	{attribute 'TcIecLibraryType'}
	{attribute 'external_name' := 'F_VN_KeyPointsGFTTExp_GUID_AB658F05_AE08_576E_4247_1E7B0BCA6233'}
	(* Detects keypoints using the GFTT method, which detects strong corners. (expert function) *)
	FUNCTION F_VN_KeyPointsGFTTExp : HRESULT
	VAR_INPUT
		ipSrcImage	:	ITcVnImage;	(* Source image *)
		ipKeyPoints	:	REFERENCE TO ITcVnContainer;	(* Returns a container which is filled with the keypoints (ContainerType_Vector_TcVnKeyPoint; Non-zero interface pointers are reused.) *)
		ipMask	:	ITcVnImage;	(* Mask to specify, where to look for keypoints (set to 0 if no mask required) *)
		stParams	:	REFERENCE TO TcVnParamsGFTT;	(* Additional expert parameters *)
		hrPrev	:	HRESULT;	(* HRESULT indicating the result of previous operations (If SUCCEEDED(hrPrev) equals false, no operation is executed.) *)
	END_VAR

END_FUNCTION

// Functions/Keypoint Features/F_VN_KeyPointsMSER

	{attribute 'TcIecLibraryType'}
	{attribute 'external_name' := 'F_VN_KeyPointsMSER_GUID_593D7D5C_CD62_5D15_521E_85C3A9A2E7E5'}
	(* Detects keypoints using the MSER method. *)
	FUNCTION F_VN_KeyPointsMSER : HRESULT
	VAR_INPUT
		ipSrcImage	:	ITcVnImage;	(* Source image *)
		ipKeyPoints	:	REFERENCE TO ITcVnContainer;	(* Returns a container which is filled with the keypoints (ContainerType_Vector_TcVnKeyPoint; Non-zero interface pointers are reused.) *)
		hrPrev	:	HRESULT;	(* HRESULT indicating the result of previous operations (If SUCCEEDED(hrPrev) equals false, no operation is executed.) *)
	END_VAR

END_FUNCTION

// Functions/Keypoint Features/F_VN_KeyPointsMSERExp

	{attribute 'TcIecLibraryType'}
	{attribute 'external_name' := 'F_VN_KeyPointsMSERExp_GUID_ABE22F08_7F3B_521F_6B7B_35024442B7CC'}
	(* Detects keypoints using the MSER method. (expert function) *)
	FUNCTION F_VN_KeyPointsMSERExp : HRESULT
	VAR_INPUT
		ipSrcImage	:	ITcVnImage;	(* Source image *)
		ipKeyPoints	:	REFERENCE TO ITcVnContainer;	(* Returns a container which is filled with the keypoints (ContainerType_Vector_TcVnKeyPoint; Non-zero interface pointers are reused.) *)
		ipMask	:	ITcVnImage;	(* Mask to specify, where to look for keypoints (set to 0 if no mask required) *)
		stParams	:	REFERENCE TO TcVnParamsMSER;	(* Additional expert parameters *)
		hrPrev	:	HRESULT;	(* HRESULT indicating the result of previous operations (If SUCCEEDED(hrPrev) equals false, no operation is executed.) *)
	END_VAR

END_FUNCTION

// Functions/Keypoint Features/F_VN_KeyPointsSB

	{attribute 'TcIecLibraryType'}
	{attribute 'external_name' := 'F_VN_KeyPointsSB_GUID_2AF0CAD1_6515_5A1D_720D_33AA4C99BB05'}
	(* Detects keypoints using a Simple Blob method:
          - several iterations apply different thresholds to source image
          - connected components (blobs) are detected
          - the center and radius of the blobs are returned as keypoints *)
	FUNCTION F_VN_KeyPointsSB : HRESULT
	VAR_INPUT
		ipSrcImage	:	ITcVnImage;	(* Source image *)
		ipKeyPoints	:	REFERENCE TO ITcVnContainer;	(* Returns a container which is filled with the keypoints (ContainerType_Vector_TcVnKeyPoint; Non-zero interface pointers are reused.) *)
		hrPrev	:	HRESULT;	(* HRESULT indicating the result of previous operations (If SUCCEEDED(hrPrev) equals false, no operation is executed.) *)
	END_VAR

END_FUNCTION

// Functions/Keypoint Features/F_VN_KeyPointsSBExp

	{attribute 'TcIecLibraryType'}
	{attribute 'external_name' := 'F_VN_KeyPointsSBExp_GUID_81F47CE7_8C3F_532C_650C_F93B4893D1D6'}
	(* 
          Detects keypoints using a Simple Blob method (expert function)
          - several iterations apply different thresholds to source image
          - connected components (blobs) are detected
          - the center and radius of the blobs are returned as keypoints
         *)
	FUNCTION F_VN_KeyPointsSBExp : HRESULT
	VAR_INPUT
		ipSrcImage	:	ITcVnImage;	(* Source image *)
		ipKeyPoints	:	REFERENCE TO ITcVnContainer;	(* Returns a container which is filled with the keypoints (ContainerType_Vector_TcVnKeyPoint; Non-zero interface pointers are reused.) *)
		ipMask	:	ITcVnImage;	(* Mask to specify, where to look for keypoints (currently not supported, set to 0) *)
		stParams	:	REFERENCE TO TcVnParamsSB;	(* Several parameters to filter the detected blobs *)
		hrPrev	:	HRESULT;	(* HRESULT indicating the result of previous operations (If SUCCEEDED(hrPrev) equals false, no operation is executed.) *)
	END_VAR

END_FUNCTION

// Functions/Keypoint Features/F_VN_MatchDescriptorsBF

	{attribute 'TcIecLibraryType'}
	{attribute 'external_name' := 'F_VN_MatchDescriptorsBF_GUID_B3966293_F5E5_53ED_7EA9_8C1C568150F9'}
	(* Match descriptors using a brute force approach. *)
	FUNCTION F_VN_MatchDescriptorsBF : HRESULT
	VAR_INPUT
		ipQueryDescriptors	:	ITcVnImage;	(* Query descriptors *)
		ipTrainDescriptors	:	ITcVnImage;	(* Training descriptors *)
		ipMatches	:	REFERENCE TO ITcVnContainer;	(* Returns a container which is filled with the descriptor matches (ContainerType_Vector_TcVnDMatch; Non-zero interface pointers are reused.) *)
		hrPrev	:	HRESULT;	(* HRESULT indicating the result of previous operations (If SUCCEEDED(hrPrev) equals false, no operation is executed.) *)
	END_VAR

END_FUNCTION

// Functions/Keypoint Features/F_VN_MatchDescriptorsBFExp

	{attribute 'TcIecLibraryType'}
	{attribute 'external_name' := 'F_VN_MatchDescriptorsBFExp_GUID_428339F2_71AA_5944_450A_B44763AAACE5'}
	(* Match descriptors using a brute force approach. (expert function) *)
	FUNCTION F_VN_MatchDescriptorsBFExp : HRESULT
	VAR_INPUT
		ipQueryDescriptors	:	ITcVnImage;	(* Query descriptors *)
		ipTrainDescriptors	:	ITcVnImage;	(* Training descriptors *)
		ipMatches	:	REFERENCE TO ITcVnContainer;	(* Returns a container which is filled with the descriptor matches (ContainerType_Vector_TcVnDMatch; Non-zero interface pointers are reused.) *)
		ipMask	:	ITcVnImage;	(* Mask to specify permissable matches, i.e. query[i] can be matched with train[j] only if mask[i][j] != 0 (set to 0 if no mask required) *)
		eNormType	:	ETcVnNormalizationType;	(* Normalization type (only L1, L2, L2SQR, HAMMING, HAMMING2 supported). HAMMING2 should be used for ORB descriptors if the ORB nBriefPoints parameter is 3 or 4) *)
		bCrossCheck	:	BOOL;	(* If true, only consistent matches are returned, i.e. query->train and train->query detect the same match *)
		hrPrev	:	HRESULT;	(* HRESULT indicating the result of previous operations (If SUCCEEDED(hrPrev) equals false, no operation is executed.) *)
	END_VAR

END_FUNCTION

// Functions/Keypoint Features/F_VN_MatchDescriptorsFlannLsh

	{attribute 'TcIecLibraryType'}
	{attribute 'external_name' := 'F_VN_MatchDescriptorsFlannLsh_GUID_6A0861D1_F3ED_5BC5_5E07_F85811927297'}
	(* Match descriptors using a FLANN based approach with LSH index. *)
	FUNCTION F_VN_MatchDescriptorsFlannLsh : HRESULT
	VAR_INPUT
		ipQueryDescriptors	:	ITcVnImage;	(* Query descriptors *)
		ipTrainDescriptors	:	ITcVnImage;	(* Training descriptors *)
		ipMatches	:	REFERENCE TO ITcVnContainer;	(* Returns a container which is filled with the descriptor matches (ContainerType_Vector_TcVnDMatch; Non-zero interface pointers are reused.) *)
		hrPrev	:	HRESULT;	(* HRESULT indicating the result of previous operations (If SUCCEEDED(hrPrev) equals false, no operation is executed.) *)
	END_VAR

END_FUNCTION

// Functions/Keypoint Features/F_VN_MatchDescriptorsFlannLshExp

	{attribute 'TcIecLibraryType'}
	{attribute 'external_name' := 'F_VN_MatchDescriptorsFlannLshExp_GUID_A6B46D94_1077_5A28_49E0_938BA5777C1C'}
	(* Match descriptors using a FLANN based approach with LSH index. (expert function) *)
	FUNCTION F_VN_MatchDescriptorsFlannLshExp : HRESULT
	VAR_INPUT
		ipQueryDescriptors	:	ITcVnImage;	(* Query descriptors *)
		ipTrainDescriptors	:	ITcVnImage;	(* Training descriptors *)
		ipMatches	:	REFERENCE TO ITcVnContainer;	(* Returns a container which is filled with the descriptor matches (ContainerType_Vector_TcVnDMatch; Non-zero interface pointers are reused.) *)
		nTableNumber	:	UDINT;	(* Number of tables *)
		nKeySize	:	UDINT;	(* Key size *)
		nMultiProbeLevel	:	UDINT;	(* Multi-probe level *)
		nChecks	:	UDINT;	(* Maximum number of visited leafs when searching for neighbors *)
		hrPrev	:	HRESULT;	(* HRESULT indicating the result of previous operations (If SUCCEEDED(hrPrev) equals false, no operation is executed.) *)
	END_VAR

END_FUNCTION

// Functions/Keypoint Features/F_VN_MatchDescriptorsKnnBF

	{attribute 'TcIecLibraryType'}
	{attribute 'external_name' := 'F_VN_MatchDescriptorsKnnBF_GUID_032847F3_E5D2_5453_7642_ACD471D5C57D'}
	(* Match descriptors (k nearest neighbors) using a brute force approach. *)
	FUNCTION F_VN_MatchDescriptorsKnnBF : HRESULT
	VAR_INPUT
		ipQueryDescriptors	:	ITcVnImage;	(* Query descriptors *)
		ipTrainDescriptors	:	ITcVnImage;	(* Training descriptors *)
		ipMatches	:	REFERENCE TO ITcVnContainer;	(* Returns a container which is filled with the descriptor matches (ContainerType_Vector_Vector_TcVnDMatch; Non-zero interface pointers are reused.) *)
		nK	:	UDINT;	(* Amount of best matches to search for *)
		hrPrev	:	HRESULT;	(* HRESULT indicating the result of previous operations (If SUCCEEDED(hrPrev) equals false, no operation is executed.) *)
	END_VAR

END_FUNCTION

// Functions/Keypoint Features/F_VN_MatchDescriptorsKnnBFExp

	{attribute 'TcIecLibraryType'}
	{attribute 'external_name' := 'F_VN_MatchDescriptorsKnnBFExp_GUID_4F5F4687_0324_5F53_4ED1_15CF466AF469'}
	(* Match descriptors (k nearest neighbors) using a brute force approach. (expert function) *)
	FUNCTION F_VN_MatchDescriptorsKnnBFExp : HRESULT
	VAR_INPUT
		ipQueryDescriptors	:	ITcVnImage;	(* Query descriptors *)
		ipTrainDescriptors	:	ITcVnImage;	(* Training descriptors *)
		ipMatches	:	REFERENCE TO ITcVnContainer;	(* Returns a container which is filled with the descriptor matches (ContainerType_Vector_Vector_TcVnDMatch; Non-zero interface pointers are reused.) *)
		nK	:	UDINT;	(* Amount of best matches to search for *)
		ipMask	:	ITcVnImage;	(* Mask to specify permissable matches, i.e. query[i] can be matched with train[j] only if mask[i][j] != 0 (set to 0 if no mask required) *)
		bCompactResult	:	BOOL;	(* If true, matches vector does not contain entries for fully masked-out query descriptors *)
		eNormType	:	ETcVnNormalizationType;	(* Normalization type (only L1, L2, L2SQR, HAMMING, HAMMING2 supported). HAMMING2 should be used for ORB descriptors if the ORB nBriefPoints parameter is 3 or 4) *)
		bCrossCheck	:	BOOL;	(* If true, only consistent matches are returned, i.e. query->train and train->query detect the same match (only used if nK = 1) *)
		hrPrev	:	HRESULT;	(* HRESULT indicating the result of previous operations (If SUCCEEDED(hrPrev) equals false, no operation is executed.) *)
	END_VAR

END_FUNCTION

// Functions/Keypoint Features/F_VN_MatchDescriptorsKnnFlannLsh

	{attribute 'TcIecLibraryType'}
	{attribute 'external_name' := 'F_VN_MatchDescriptorsKnnFlannLsh_GUID_C8244361_8A2E_5422_786B_9C4704343BF2'}
	(* Match descriptors (k nearest neighbors) using a FLANN based approach with LSH index. *)
	FUNCTION F_VN_MatchDescriptorsKnnFlannLsh : HRESULT
	VAR_INPUT
		ipQueryDescriptors	:	ITcVnImage;	(* Query descriptors *)
		ipTrainDescriptors	:	ITcVnImage;	(* Training descriptors *)
		ipMatches	:	REFERENCE TO ITcVnContainer;	(* Returns a container which is filled with the descriptor matches (ContainerType_Vector_Vector_TcVnDMatch; Non-zero interface pointers are reused.) *)
		nK	:	UDINT;	(* Amount of best matches to search for *)
		hrPrev	:	HRESULT;	(* HRESULT indicating the result of previous operations (If SUCCEEDED(hrPrev) equals false, no operation is executed.) *)
	END_VAR

END_FUNCTION

// Functions/Keypoint Features/F_VN_MatchDescriptorsKnnFlannLshExp

	{attribute 'TcIecLibraryType'}
	{attribute 'external_name' := 'F_VN_MatchDescriptorsKnnFlannLshExp_GUID_C49C1B5A_C1AC_5443_653F_891B8408EDAA'}
	(* Match descriptors (k nearest neighbors) using a FLANN based approach with LSH index. (expert function) *)
	FUNCTION F_VN_MatchDescriptorsKnnFlannLshExp : HRESULT
	VAR_INPUT
		ipQueryDescriptors	:	ITcVnImage;	(* Query descriptors *)
		ipTrainDescriptors	:	ITcVnImage;	(* Training descriptors *)
		ipMatches	:	REFERENCE TO ITcVnContainer;	(* Returns a container which is filled with the descriptor matches (ContainerType_Vector_Vector_TcVnDMatch; Non-zero interface pointers are reused.) *)
		nK	:	UDINT;	(* Amount of best matches to search for *)
		nTableNumber	:	UDINT;	(* Number of tables *)
		nKeySize	:	UDINT;	(* Key size *)
		nMultiProbeLevel	:	UDINT;	(* Multi-probe level *)
		nChecks	:	UDINT;	(* Maximum number of visited leafs when searching for neighbors *)
		hrPrev	:	HRESULT;	(* HRESULT indicating the result of previous operations (If SUCCEEDED(hrPrev) equals false, no operation is executed.) *)
	END_VAR

END_FUNCTION

// Functions/Keypoint Features/F_VN_RegionsMSER

	{attribute 'TcIecLibraryType'}
	{attribute 'external_name' := 'F_VN_RegionsMSER_GUID_55741E50_BE33_5462_61F4_4C1E00297C7D'}
	(* Detects regions using the MSER method. *)
	FUNCTION F_VN_RegionsMSER : HRESULT
	VAR_INPUT
		ipSrcImage	:	ITcVnImage;	(* Source image *)
		ipRegions	:	REFERENCE TO ITcVnContainer;	(* Returns a container which is filled with the region points (ContainerType_Vector_Vector_TcVnPoint2_DINT; Non-zero interface pointers are reused.) *)
		ipBoundingBoxes	:	REFERENCE TO ITcVnContainer;	(* Returns a container which is filled with the region bounding boxes (ContainerType_Vector_TcVnRectangle_DINT; Non-zero interface pointers are reused.) *)
		hrPrev	:	HRESULT;	(* HRESULT indicating the result of previous operations (If SUCCEEDED(hrPrev) equals false, no operation is executed.) *)
	END_VAR

END_FUNCTION

// Functions/Keypoint Features/F_VN_RegionsMSERExp

	{attribute 'TcIecLibraryType'}
	{attribute 'external_name' := 'F_VN_RegionsMSERExp_GUID_E4887BE5_69AC_5ABE_40D6_3515223EBD0A'}
	(* Detects regions using the MSER method. (expert function) *)
	FUNCTION F_VN_RegionsMSERExp : HRESULT
	VAR_INPUT
		ipSrcImage	:	ITcVnImage;	(* Source image *)
		ipRegions	:	REFERENCE TO ITcVnContainer;	(* Returns a container which is filled with the region points (ContainerType_Vector_Vector_TcVnPoint2_DINT; Non-zero interface pointers are reused.) *)
		ipBoundingBoxes	:	REFERENCE TO ITcVnContainer;	(* Returns a container which is filled with the region bounding boxes (ContainerType_Vector_TcVnRectangle_DINT; Non-zero interface pointers are reused.) *)
		stParams	:	REFERENCE TO TcVnParamsMSER;	(* Additional expert parameters *)
		hrPrev	:	HRESULT;	(* HRESULT indicating the result of previous operations (If SUCCEEDED(hrPrev) equals false, no operation is executed.) *)
	END_VAR

END_FUNCTION

// Functions/Code Reading/F_VN_ReadBarcode

	{attribute 'TcIecLibraryType'}
	{attribute 'external_name' := 'F_VN_ReadBarcode_GUID_7EE00F83_82CC_5410_5E28_06AA8744DAB0'}
	(* Detect and interpret a 1d barcode within the provided image.
          Can be canceled by Watchdog. *)
	FUNCTION F_VN_ReadBarcode : HRESULT
	VAR_INPUT
		ipSrcImage	:	ITcVnImage;	(* Source image (USINT elements, 1 channel or 3 channel (3 channel input is expected to be RGB and internally converted to Gray)) *)
		ipDecodedData	:	REFERENCE TO ITcVnContainer;	(* Returns the decoded code (ContainerType_Vector_String_SINT) *)
		eBarcodeType	:	UDINT;	(* Types of barcode to search for (ETcVnBarcodeType) *)
		hrPrev	:	HRESULT;	(* HRESULT indicating the result of previous operations (If SUCCEEDED(hrPrev) equals false, no operation is executed.) *)
	END_VAR

END_FUNCTION

// Functions/Code Reading/F_VN_ReadBarcodeExp

	{attribute 'TcIecLibraryType'}
	{attribute 'external_name' := 'F_VN_ReadBarcodeExp_GUID_746E9938_9353_5E2C_6CDD_CD6CAD35E403'}
	(* Detect and interpret a 1d barcode within the provided image.
          Can be canceled by Watchdog. *)
	FUNCTION F_VN_ReadBarcodeExp : HRESULT
	VAR_INPUT
		ipSrcImage	:	ITcVnImage;	(* Source image (USINT elements, 1 channel or 3 channel (3 channel input is expected to be RGB and internally converted to Gray)) *)
		ipDecodedData	:	REFERENCE TO ITcVnContainer;	(* Returns the decoded code (ContainerType_Vector_String_SINT) *)
		ipContours	:	REFERENCE TO ITcVnContainer;	(* Returns the code positions as contours (ContainerType_Vector_Vector_TcVnPoint2_DINT) *)
		eBarcodeType	:	UDINT;	(* Types of barcode to search for (ETcVnBarcodeType) *)
		nCodeNumber	:	DINT;	(* Number of 1d barcode that should be detected within the provided image (currently only 1 supported). *)
		eSearchDirection	:	ETcVnBarcodeSearchDirection;	(* Barcode search direction. *)
		hrPrev	:	HRESULT;	(* HRESULT indicating the result of previous operations (If SUCCEEDED(hrPrev) equals false, no operation is executed.) *)
	END_VAR

END_FUNCTION

// Functions/Code Reading/F_VN_ReadDataMatrixCode

	{attribute 'TcIecLibraryType'}
	{attribute 'external_name' := 'F_VN_ReadDataMatrixCode_GUID_B4511350_6021_5C04_7D51_7B88C8EE3F13'}
	(* Detect and interpret a data matrix code within the provided image. *)
	FUNCTION F_VN_ReadDataMatrixCode : HRESULT
	VAR_INPUT
		ipSrcImage	:	ITcVnImage;	(* Source image (USINT elements, 1 or 3 channels) *)
		ipDecodedData	:	REFERENCE TO ITcVnContainer;	(* Returns the decoded code (ContainerType_Vector_String_SINT) *)
		hrPrev	:	HRESULT;	(* HRESULT indicating the result of previous operations (If SUCCEEDED(hrPrev) equals false, no operation is executed.) *)
	END_VAR

END_FUNCTION

// Functions/Code Reading/F_VN_ReadDataMatrixCodeExp

	{attribute 'TcIecLibraryType'}
	{attribute 'external_name' := 'F_VN_ReadDataMatrixCodeExp_GUID_2A0AE396_48EA_536D_5539_B99ADA95FFAB'}
	(* Detect and interpret a data matrix code within the provided image. *)
	FUNCTION F_VN_ReadDataMatrixCodeExp : HRESULT
	VAR_INPUT
		ipSrcImage	:	ITcVnImage;	(* Source image (USINT elements, 1 or 3 channels) *)
		ipDecodedData	:	REFERENCE TO ITcVnContainer;	(* Returns the decoded code (ContainerType_Vector_String_SINT) *)
		ipContours	:	REFERENCE TO ITcVnContainer;	(* Returns the code positions as contours (ContainerType_Vector_Vector_TcVnPoint2_DINT) *)
		nCodeNumber	:	DINT;	(* Number of data matrix codes that should be detected within the provided image. (If set to -1, it is tried to detect all data matrix codes.) *)
		eSearchStrategy	:	UDINT;	(* Used search strategy (ETcVn2dCodeSearchStrategy) *)
		hrPrev	:	HRESULT;	(* HRESULT indicating the result of previous operations (If SUCCEEDED(hrPrev) equals false, no operation is executed.) *)
	END_VAR

END_FUNCTION

// Functions/Code Reading/F_VN_ReadPharmaCode

	{attribute 'TcIecLibraryType'}
	{attribute 'external_name' := 'F_VN_ReadPharmaCode_GUID_E6E75064_05CB_51B6_5B74_A32B7C745647'}
	(* Detect and interpret a pharma code within the provided image.
				Can be canceled by Watchdog. *)
	FUNCTION F_VN_ReadPharmaCode : HRESULT
	VAR_INPUT
		ipSrcImage	:	ITcVnImage;	(* Source image (1 channel (all element types) or 3 channel with elements of type TCVN_ET_USINT, TCVN_ET_UINT or TCVN_ET_REAL (3 channel input is expected to be RGB and internally converted to Gray)) *)
		ipDecodedData	:	REFERENCE TO ITcVnContainer;	(* Returns the decoded code (ContainerType_Vector_String_SINT) *)
		hrPrev	:	HRESULT;	(* HRESULT indicating the result of previous operations (If SUCCEEDED(hrPrev) equals false, no operation is executed.) *)
	END_VAR

END_FUNCTION

// Functions/Code Reading/F_VN_ReadPharmaCodeExp

	{attribute 'TcIecLibraryType'}
	{attribute 'external_name' := 'F_VN_ReadPharmaCodeExp_GUID_E3F97547_DCBF_56B5_54C9_CF3A6BD2500C'}
	(* Detect and interpret a pharma code within the provided image.
				Can be canceled by Watchdog. *)
	FUNCTION F_VN_ReadPharmaCodeExp : HRESULT
	VAR_INPUT
		ipSrcImage	:	ITcVnImage;	(* Source image (1 channel (all element types) or 3 channel with elements of type TCVN_ET_USINT, TCVN_ET_UINT or TCVN_ET_REAL (3 channel input is expected to be RGB and internally converted to Gray)) *)
		ipDecodedData	:	REFERENCE TO ITcVnContainer;	(* Returns the decoded code (ContainerType_Vector_String_SINT) *)
		ipContours	:	REFERENCE TO ITcVnContainer;	(* Returns the code positions as contours (ContainerType_Vector_Vector_TcVnPoint2_DINT) *)
		nCodeNumber	:	DINT;	(* Number of pharma codes that should be detected within the provided image (currently only 1 supported). *)
		nMinBarNumber	:	INT;	(* Minimal number of (dark) bars that codes must have. *)
		hrPrev	:	HRESULT;	(* HRESULT indicating the result of previous operations (If SUCCEEDED(hrPrev) equals false, no operation is executed.) *)
	END_VAR

END_FUNCTION

// Functions/Code Reading/F_VN_ReadQRCode

	{attribute 'TcIecLibraryType'}
	{attribute 'external_name' := 'F_VN_ReadQRCode_GUID_61B83291_17E3_5A76_70AE_70467F2D3B85'}
	(* Detect and interpret a QR code within the provided image.
          Can be canceled by Watchdog. *)
	FUNCTION F_VN_ReadQRCode : HRESULT
	VAR_INPUT
		ipSrcImage	:	ITcVnImage;	(* Source image (USINT elements, 1 channel or 3 channel (3 channel input is expected to be RGB and internally converted to Gray)) *)
		ipDecodedData	:	REFERENCE TO ITcVnContainer;	(* Returns the decoded code (ContainerType_Vector_String_SINT) *)
		hrPrev	:	HRESULT;	(* HRESULT indicating the result of previous operations (If SUCCEEDED(hrPrev) equals false, no operation is executed.) *)
	END_VAR

END_FUNCTION

// Functions/Code Reading/F_VN_ReadQRCodeExp

	{attribute 'TcIecLibraryType'}
	{attribute 'external_name' := 'F_VN_ReadQRCodeExp_GUID_EC08C934_0AC5_5C4F_7BC3_2B90FBC1E2D7'}
	(* Detect and interpret a QR code within the provided image.
          Can be canceled by Watchdog. *)
	FUNCTION F_VN_ReadQRCodeExp : HRESULT
	VAR_INPUT
		ipSrcImage	:	ITcVnImage;	(* Source image (USINT elements, 1 channel or 3 channel (3 channel input is expected to be RGB and internally converted to Gray)) *)
		ipDecodedData	:	REFERENCE TO ITcVnContainer;	(* Returns the decoded code (ContainerType_Vector_String_SINT) *)
		ipContours	:	REFERENCE TO ITcVnContainer;	(* Returns the code positions as contours (ContainerType_Vector_Vector_TcVnPoint2_DINT) *)
		nCodeNumber	:	DINT;	(* Number of QR codes that should be detected within the provided image (currently only 1 supported). *)
		eSearchStrategy	:	UDINT;	(* Used search strategy (ETcVn2dCodeSearchStrategy) *)
		hrPrev	:	HRESULT;	(* HRESULT indicating the result of previous operations (If SUCCEEDED(hrPrev) equals false, no operation is executed.) *)
	END_VAR

END_FUNCTION

// Functions/Image Analysis/Object Detection/F_VN_AdjustActiveContour

	{attribute 'TcIecLibraryType'}
	{attribute 'external_name' := 'F_VN_AdjustActiveContour_GUID_74BDF730_EC57_5A0C_4BC7_A5964F056D8C'}
	(* Adjust active contour (snake) in order to minimize its cummulative (internal and external) energy. *)
	FUNCTION F_VN_AdjustActiveContour : HRESULT
	VAR_INPUT
		ipImage	:	ITcVnImage;	(* Source image (1 channel, USINT elements) *)
		ipActiveContour	:	ITcVnContainer;	(* Initial contour, which will be adjusted *)
		fAlpha	:	REAL;	(* Continuity energy coefficient *)
		fBeta	:	REAL;	(* Curvature energy coefficient *)
		fGamma	:	REAL;	(* Image energy coefficient *)
		nWindowWidth	:	UDINT;	(* Windows width (3, 5, 7, ...) *)
		nWindowHeight	:	UDINT;	(* Windows height (3, 5, 7, ...) *)
		nMaxIterations	:	UDINT;	(* Maximum iterations *)
		bUseGradient	:	BOOL;	(* If true, the gradient magnitude is used as image energy (otherwise: pixel intensity) *)
		hrPrev	:	HRESULT;	(* HRESULT indicating the result of previous operations (If SUCCEEDED(hrPrev) equals false, no operation is executed.) *)
	END_VAR

END_FUNCTION

// Functions/Image Analysis/Object Detection/F_VN_DetectBlobs

	{attribute 'TcIecLibraryType'}
	{attribute 'external_name' := 'F_VN_DetectBlobs_GUID_457E40D7_8624_5A85_76C5_7324B3EA04E5'}
	(* Detects blob-contours. Applies a threshold, a contour search and offers several options for filtering the found contours. Provides easy setup for multiple thresholds and combination of results. *)
	FUNCTION F_VN_DetectBlobs : HRESULT
	VAR_INPUT
		ipSrcImage	:	ITcVnImage;	(* Source image (USINT or REAL, 1 channel or 3 channel (3 channel input is expected to be RGB and internally converted to Gray)) *)
		ipBlobContours	:	REFERENCE TO ITcVnContainer;	(* Returns a container which is filled with the found contours (ContainerType_Vector_Vector_TcVnPoint2_DINT; The elements of this container are single contours. Non-zero interface pointers are reused.) *)
		stParams	:	REFERENCE TO TcVnParamsBlobDetection;	(* Parameters to filter the detected contours. *)
		hrPrev	:	HRESULT;	(* HRESULT indicating the result of previous operations (If SUCCEEDED(hrPrev) equals false, no operation is executed.) *)
	END_VAR

END_FUNCTION

// Functions/Image Analysis/Object Detection/F_VN_DetectBlobsExp

	{attribute 'TcIecLibraryType'}
	{attribute 'external_name' := 'F_VN_DetectBlobsExp_GUID_6004E0FE_504F_5A15_5C72_A38ABCE1764F'}
	(* Detects blob-contours. Applies a threshold, a contour search and offers several options for filtering the found contours. Provides easy setup for multiple thresholds and combination of results. (expert function) *)
	FUNCTION F_VN_DetectBlobsExp : HRESULT
	VAR_INPUT
		ipSrcImage	:	ITcVnImage;	(* Source image (USINT or REAL, 1 channel or 3 channel (3 channel input is expected to be RGB and internally converted to Gray)) *)
		ipBlobContours	:	REFERENCE TO ITcVnContainer;	(* Returns a container which is filled with the found contours (ContainerType_Vector_Vector_TcVnPoint2_DINT; The elements of this container are single contours. Non-zero interface pointers are reused.) *)
		stParams	:	REFERENCE TO TcVnParamsBlobDetection;	(* Parameters to filter the detected contours. *)
		aOffset	:	REFERENCE TO TcVnPoint;	(* Offset by which every contour point is shifted *)
		hrPrev	:	HRESULT;	(* HRESULT indicating the result of previous operations (If SUCCEEDED(hrPrev) equals false, no operation is executed.) *)
	END_VAR

END_FUNCTION

// Functions/Image Analysis/Object Detection/F_VN_FindContourHierarchyExp

	{attribute 'TcIecLibraryType'}
	{attribute 'external_name' := 'F_VN_FindContourHierarchyExp_GUID_08667274_4195_59C8_59FC_347C933C80CD'}
	(* Search for object contours in a binary image and determine their hierarchical relationship. (expert function) *)
	FUNCTION F_VN_FindContourHierarchyExp : HRESULT
	VAR_INPUT
		ipSrcImage	:	ITcVnImage;	(* Source image (1 channel, binary) *)
		ipContours	:	REFERENCE TO ITcVnContainer;	(* Returns a container which is filled with the found contours (ContainerType_Vector_Vector_TcVnPoint2_DINT; The elements of this container are single contours. Non-zero interface pointers are reused.) *)
		ipHierarchy	:	REFERENCE TO ITcVnContainer;	(* Returns a container which is filled with information on the found contours' hierarchy (ContainerType_Vector_TcVnVector4_DINT; The elements of this container are four-dimensional vectors containing the 0-based indices of the next [0] and the previous contour [1] at the same level, the first child [2], and the parent [3]. Non-zero interface pointers are reused.) *)
		eRetrievalMode	:	ETcVnContourRetrievalMode;	(* Specifies which contours are retrieved and how their relationship is encoded *)
		eApproximationMethod	:	ETcVnContourApproximationMethod;	(* Contour encoding *)
		aOffset	:	REFERENCE TO TcVnPoint;	(* Offset by which every contour point is shifted *)
		hrPrev	:	HRESULT;	(* HRESULT indicating the result of previous operations (If SUCCEEDED(hrPrev) equals false, no operation is executed.) *)
	END_VAR

END_FUNCTION

// Functions/Image Analysis/Object Detection/F_VN_FindContours

	{attribute 'TcIecLibraryType'}
	{attribute 'external_name' := 'F_VN_FindContours_GUID_60AD5F03_F669_5AFB_6F67_9C388BC37A3E'}
	(* Search for object contours in a binary image. Returns only external contours. *)
	FUNCTION F_VN_FindContours : HRESULT
	VAR_INPUT
		ipSrcImage	:	ITcVnImage;	(* Source image (1 channel, binary) *)
		ipContours	:	REFERENCE TO ITcVnContainer;	(* Returns a container which is filled with the found contours (ContainerType_Vector_Vector_TcVnPoint2_DINT; The elements of this container are single contours. Non-zero interface pointers are reused.) *)
		hrPrev	:	HRESULT;	(* HRESULT indicating the result of previous operations (If SUCCEEDED(hrPrev) equals false, no operation is executed.) *)
	END_VAR

END_FUNCTION

// Functions/Image Analysis/Object Detection/F_VN_FindContoursExp

	{attribute 'TcIecLibraryType'}
	{attribute 'external_name' := 'F_VN_FindContoursExp_GUID_10AF9C9F_9D33_58ED_4B7C_62A006BC4250'}
	(* Search for object contours in a binary image. (expert function) *)
	FUNCTION F_VN_FindContoursExp : HRESULT
	VAR_INPUT
		ipSrcImage	:	ITcVnImage;	(* Source image (1 channel, binary) *)
		ipContours	:	REFERENCE TO ITcVnContainer;	(* Returns a container which is filled with the found contours (ContainerType_Vector_Vector_TcVnPoint2_DINT; The elements of this container are single contours. Non-zero interface pointers are reused.) *)
		eRetrievalMode	:	ETcVnContourRetrievalMode;	(* Specifies which contours are retrieved and how their relationship is encoded *)
		eApproximationMethod	:	ETcVnContourApproximationMethod;	(* Contour encoding *)
		aOffset	:	REFERENCE TO TcVnPoint;	(* Offset by which every contour point is shifted *)
		hrPrev	:	HRESULT;	(* HRESULT indicating the result of previous operations (If SUCCEEDED(hrPrev) equals false, no operation is executed.) *)
	END_VAR

END_FUNCTION

// Functions/Image Analysis/Object Detection/F_VN_HoughCircles

	{attribute 'TcIecLibraryType'}
	{attribute 'external_name' := 'F_VN_HoughCircles_GUID_5A3C1972_E2A2_5BE7_7B88_6638F06E8880'}
	(* Search for circles using the Hough transform. *)
	FUNCTION F_VN_HoughCircles : HRESULT
	VAR_INPUT
		ipSrcImage	:	ITcVnImage;	(* Source image (USINT, 1 channel, gray-level) *)
		ipCircles	:	REFERENCE TO ITcVnContainer;	(* Returns a container which is filled with the found circles (ContainerType_Vector_TcVnVector3_REAL; Each container element contains the x coordinate of the circle center [0], the y coordinate of the circle center [1], and the radius [2], respectively. Non-zero interface pointers are reused.) *)
		fInvAccuRatio	:	LREAL;	(* Inverted ratio of the accumulator size in relation to the source image's size (must be > 0. A value of 2 means that the size is halved in both directions.) *)
		fMinDist	:	LREAL;	(* Smallest allowed distance of two circles (must be > 0) *)
		hrPrev	:	HRESULT;	(* HRESULT indicating the result of previous operations (If SUCCEEDED(hrPrev) equals false, no operation is executed.) *)
	END_VAR

END_FUNCTION

// Functions/Image Analysis/Object Detection/F_VN_HoughCirclesExp

	{attribute 'TcIecLibraryType'}
	{attribute 'external_name' := 'F_VN_HoughCirclesExp_GUID_6D107BB0_0DB4_5005_6438_B72FFE9DD6B5'}
	(* Search for circles using the Hough transform. (expert function) *)
	FUNCTION F_VN_HoughCirclesExp : HRESULT
	VAR_INPUT
		ipSrcImage	:	ITcVnImage;	(* Source image (USINT, 1 channel, gray-level) *)
		ipCircles	:	REFERENCE TO ITcVnContainer;	(* Returns a container which is filled with the found circles (ContainerType_Vector_TcVnVector3_REAL; Each container element contains the x coordinate of the circle center [0], the y coordinate of the circle center [1], and the radius [2], respectively. Non-zero interface pointers are reused.) *)
		fInvAccuRatio	:	LREAL;	(* Inverted ratio of the accumulator size in relation to the source image's size (must be > 0. A value of 2 means that the size is halved in both directions.) *)
		fMinDist	:	LREAL;	(* Smallest allowed distance of two circles (must be > 0) *)
		eHoughMethod	:	ETcVnHoughMethod;	(* Hough method to use (currently only valid value: GRADIENT) *)
		fParam1	:	LREAL;	(* First method specific parameter (GRADIENT: upper threshold for canny edge detection, which must be > 0) *)
		fParam2	:	LREAL;	(* Second method specific parameter (GRADIENT: accumulator threshold for detecting circle centers, which must be > 0) *)
		nMinRadius	:	UDINT;	(* Minimum circle radius allowed *)
		nMaxRadius	:	UDINT;	(* Maximum circle radius allowed (if 0, the value is internally set to max(image rows, image columns)) *)
		hrPrev	:	HRESULT;	(* HRESULT indicating the result of previous operations (If SUCCEEDED(hrPrev) equals false, no operation is executed.) *)
	END_VAR

END_FUNCTION

// Functions/Image Analysis/Object Detection/F_VN_HoughLines

	{attribute 'TcIecLibraryType'}
	{attribute 'external_name' := 'F_VN_HoughLines_GUID_EA8DF545_06D1_573B_6149_330F6A13A330'}
	(* Search for lines using the standard Hough transform. *)
	FUNCTION F_VN_HoughLines : HRESULT
	VAR_INPUT
		ipSrcImage	:	ITcVnImage;	(* Source image (USINT, 1 channel, binary, may be modified by the function) *)
		ipLines	:	REFERENCE TO ITcVnContainer;	(* Returns a container which is filled with the found lines (ContainerType_Vector_TcVnVector2_REAL; Each container element contains the distance from the origin [0] in pixels and the rotation angle [1] in radians, respectively. Non-zero interface pointers are reused.) *)
		fDistRes	:	LREAL;	(* Distance resolution of the accumulator (in pixels, must be > 0) *)
		fAngleRes	:	LREAL;	(* Angle resolution of the accumulator (in radians, must be > 0) *)
		nAccuThreshold	:	UDINT;	(* Accumulator threshold *)
		hrPrev	:	HRESULT;	(* HRESULT indicating the result of previous operations (If SUCCEEDED(hrPrev) equals false, no operation is executed.) *)
	END_VAR

END_FUNCTION

// Functions/Image Analysis/Object Detection/F_VN_HoughLinesExp

	{attribute 'TcIecLibraryType'}
	{attribute 'external_name' := 'F_VN_HoughLinesExp_GUID_C053D90B_9429_56A9_7C22_F1CD18038900'}
	(* Search for lines using the standard Hough transform. (expert function) *)
	FUNCTION F_VN_HoughLinesExp : HRESULT
	VAR_INPUT
		ipSrcImage	:	ITcVnImage;	(* Source image (USINT, 1 channel, binary, may be modified by the function) *)
		ipLines	:	REFERENCE TO ITcVnContainer;	(* Returns a container which is filled with the found lines (ContainerType_Vector_TcVnVector2_REAL; Each container element contains the distance from the origin [0] in pixels and the rotation angle [1] in radians, respectively. Non-zero interface pointers are reused.) *)
		fDistRes	:	LREAL;	(* Distance resolution of the accumulator (in pixels, must be > 0) *)
		fAngleRes	:	LREAL;	(* Angle resolution of the accumulator (in radians, must be > 0) *)
		nAccuThreshold	:	UDINT;	(* Accumulator threshold *)
		fDistResDiv	:	LREAL;	(* Divisor of the distance resolution for the multi-scale Hough transform (>= 0, must be > 0 if fAngleResDiv is > 0) *)
		fAngleResDiv	:	LREAL;	(* Divisor of the angle resolution for the multi-scale Hough transform (>= 0, must be > 0 if fDistResDiv is > 0) *)
		hrPrev	:	HRESULT;	(* HRESULT indicating the result of previous operations (If SUCCEEDED(hrPrev) equals false, no operation is executed.) *)
	END_VAR

END_FUNCTION

// Functions/Image Analysis/Object Detection/F_VN_HoughLinesP

	{attribute 'TcIecLibraryType'}
	{attribute 'external_name' := 'F_VN_HoughLinesP_GUID_3E906962_C5DF_5C0F_5FEA_7FC1FBF7BFA9'}
	(* Search for line segments using the probabilistic Hough transform. *)
	FUNCTION F_VN_HoughLinesP : HRESULT
	VAR_INPUT
		ipSrcImage	:	ITcVnImage;	(* Source image (USINT, 1 channel, binary, may be modified by the function) *)
		ipLines	:	REFERENCE TO ITcVnContainer;	(* Returns a container which is filled with the found line segments (ContainerType_Vector_TcVnVector4_DINT; Each container element contains the two ending points. Non-zero interface pointers are reused.) *)
		fDistRes	:	LREAL;	(* Distance resolution of the accumulator (in pixels, must be > 0) *)
		fAngleRes	:	LREAL;	(* Angle resolution of the accumulator (in radians, must be > 0) *)
		nAccuThreshold	:	UDINT;	(* Accumulator threshold *)
		hrPrev	:	HRESULT;	(* HRESULT indicating the result of previous operations (If SUCCEEDED(hrPrev) equals false, no operation is executed.) *)
	END_VAR

END_FUNCTION

// Functions/Image Analysis/Object Detection/F_VN_HoughLinesPExp

	{attribute 'TcIecLibraryType'}
	{attribute 'external_name' := 'F_VN_HoughLinesPExp_GUID_B3F90F27_2FE0_5D42_7B16_826EA95B9B9B'}
	(* Search for line segments using the probabilistic Hough transform. (expert function) *)
	FUNCTION F_VN_HoughLinesPExp : HRESULT
	VAR_INPUT
		ipSrcImage	:	ITcVnImage;	(* Source image (USINT, 1 channel, binary, may be modified by the function) *)
		ipLines	:	REFERENCE TO ITcVnContainer;	(* Returns a container which is filled with the found line segments (ContainerType_Vector_TcVnVector4_DINT; Each container element contains the two ending points. Non-zero interface pointers are reused.) *)
		fDistRes	:	LREAL;	(* Distance resolution of the accumulator (in pixels, must be > 0) *)
		fAngleRes	:	LREAL;	(* Angle resolution of the accumulator (in radians, must be > 0) *)
		nAccuThreshold	:	UDINT;	(* Accumulator threshold *)
		fMinLineLength	:	LREAL;	(* Minimum line length to search for *)
		fMaxLineGap	:	LREAL;	(* Maximum gap between points on the same line *)
		hrPrev	:	HRESULT;	(* HRESULT indicating the result of previous operations (If SUCCEEDED(hrPrev) equals false, no operation is executed.) *)
	END_VAR

END_FUNCTION

// Functions/Image Analysis/Object Detection/F_VN_MatchImageHuMoments

	{attribute 'TcIecLibraryType'}
	{attribute 'external_name' := 'F_VN_MatchImageHuMoments_GUID_0DB8C398_A80A_5CEF_7224_6E9B9FE0E9BC'}
	(* Compare two images using the Hu moment invariants. *)
	FUNCTION F_VN_MatchImageHuMoments : HRESULT
	VAR_INPUT
		ipImage1	:	ITcVnImage;	(* First image (1 channel) *)
		ipImage2	:	ITcVnImage;	(* Second image (1 channel) *)
		eComparisonMethod	:	ETcVnContoursMatchComparisonMethod;	(* Method used for comparing the Hu moment invariants of the images *)
		fDissimilarity	:	REFERENCE TO LREAL;	(* Returns the dissimilarity of the image Hu moment invariants depending on the chosen comparison method *)
		hrPrev	:	HRESULT;	(* HRESULT indicating the result of previous operations (If SUCCEEDED(hrPrev) equals false, no operation is executed.) *)
	END_VAR

END_FUNCTION

// Functions/Image Analysis/Object Detection/F_VN_MatchTemplate

	{attribute 'TcIecLibraryType'}
	{attribute 'external_name' := 'F_VN_MatchTemplate_GUID_A8D71B56_095E_59D2_73F6_CCB2C3BE74F3'}
	(* Match a template image with every location in the source image (using the TCVN_TMM_CCORR_NORMED method) and save the comparison results. *)
	FUNCTION F_VN_MatchTemplate : HRESULT
	VAR_INPUT
		ipSrcImage	:	ITcVnImage;	(* Source image (USINT or REAL, 1 or 3 channels) *)
		ipTemplateImage	:	ITcVnImage;	(* Template image (same type as ipSrcImage, smaller width and height) *)
		ipResultImage	:	REFERENCE TO ITcVnImage;	(* Returns the result image (REAL, normalized to [0..1], 1 channel, dimensions: (ipSrcImage.width - ipTemplateImage.width + 1) x (ipSrcImage.height - ipTemplateImage.height + 1). The best match is the global maximum. The position in ipResultImage is the top-left corner of ipTemplateImage position in ipSrcImage) *)
		hrPrev	:	HRESULT;	(* HRESULT indicating the result of previous operations (If SUCCEEDED(hrPrev) equals false, no operation is executed.) *)
	END_VAR

END_FUNCTION

// Functions/Image Analysis/Object Detection/F_VN_MatchTemplateExp

	{attribute 'TcIecLibraryType'}
	{attribute 'external_name' := 'F_VN_MatchTemplateExp_GUID_5EBC2CC0_278B_5B6F_4801_4D5B81D6E14C'}
	(* Match a template image with every location in the source image and save the comparison results. (expert function) *)
	FUNCTION F_VN_MatchTemplateExp : HRESULT
	VAR_INPUT
		ipSrcImage	:	ITcVnImage;	(* Source image (USINT or REAL, 1 or 3 channels) *)
		ipTemplateImage	:	ITcVnImage;	(* Template image (same type as ipSrcImage, smaller width and height) *)
		ipResultImage	:	REFERENCE TO ITcVnImage;	(* Returns the result image (REAL, 1 channel, dimensions: (ipSrcImage.width - ipTemplateImage.width + 1) x (ipSrcImage.height - ipTemplateImage.height + 1). The best match is the global minimum (SQDIFF(_NORMED)) or maximum (CCORR(_NORMED), CCOEFF(_NORMED)). The position in ipResultImage is the top-left corner of ipTemplateImage position in ipSrcImage) *)
		eMatchMethod	:	ETcVnTemplateMatchMethod;	(* Specifies the template match method *)
		ipTemplateMask	:	ITcVnImage;	(* Optional mask for ipTemplateImage (only supported for SQDIFF and CCORR_NORMED, same type and size as ipTemplateImage) *)
		hrPrev	:	HRESULT;	(* HRESULT indicating the result of previous operations (If SUCCEEDED(hrPrev) equals false, no operation is executed.) *)
	END_VAR

END_FUNCTION

// Functions/Image Analysis/Object Detection/F_VN_MatchTemplateAndEvaluate

	{attribute 'TcIecLibraryType'}
	{attribute 'external_name' := 'F_VN_MatchTemplateAndEvaluate_GUID_BCAA9657_0559_5BCD_72A3_483E99CAF163'}
	(* Match a template image with every location in the source image (using the TCVN_TMM_CCORR_NORMED method) and evaluate the comparison results. Returns a sorted list of possible matches (best match first). *)
	FUNCTION F_VN_MatchTemplateAndEvaluate : HRESULT
	VAR_INPUT
		ipSrcImage	:	ITcVnImage;	(* Source image (USINT or REAL, 1 or 3 channels) *)
		ipTemplateImage	:	ITcVnImage;	(* Template image (same type as ipSrcImage, smaller width and height) *)
		ipMatches	:	REFERENCE TO ITcVnContainer;	(* Returns the matching positions (ContainerType_Vector_TcVnPoint2_DINT, where each element represents the top-left corner of ipTemplateImage) in ipSrcImage, sorted by relevance (best match first) *)
		fMatchThreshold	:	REAL;	(* Threshold to separate relevant from irrelevant matches (0..1, 1.0  would be a perfect match. To find a suitable value, you could evaluate some sample result images of F_VN_MatchTemplate.) *)
		hrPrev	:	HRESULT;	(* HRESULT indicating the result of previous operations (If SUCCEEDED(hrPrev) equals false, no operation is executed.) *)
	END_VAR

END_FUNCTION

// Functions/Image Analysis/Object Detection/F_VN_MatchTemplateAndEvaluateExp

	{attribute 'TcIecLibraryType'}
	{attribute 'external_name' := 'F_VN_MatchTemplateAndEvaluateExp_GUID_3A43F904_AE6B_5997_4A68_D3FC09A55DD2'}
	(* Match a template image with every location in the source image and evaluate the comparison results. Returns a sorted list of possible matches (best match first). (expert function) *)
	FUNCTION F_VN_MatchTemplateAndEvaluateExp : HRESULT
	VAR_INPUT
		ipSrcImage	:	ITcVnImage;	(* Source image (USINT or REAL, 1 or 3 channels) *)
		ipTemplateImage	:	ITcVnImage;	(* Template image (same type as ipSrcImage, smaller width and height) *)
		ipMatches	:	REFERENCE TO ITcVnContainer;	(* Returns the matching positions (ContainerType_Vector_TcVnPoint2_DINT, where each element represents the top-left corner of ipTemplateImage) in ipSrcImage, sorted by relevance (best match first) *)
		fMatchThreshold	:	REAL;	(* Threshold to separate relevant from irrelevant matches (0..1 for NORMED methods, otherwise dependent on template size and content. To find a suitable value, you could evaluate some sample result images of F_VN_MatchTemplateExp.) *)
		eMatchMethod	:	ETcVnTemplateMatchMethod;	(* Specifies the template match method *)
		ipTemplateMask	:	ITcVnImage;	(* Optional mask for ipTemplateImage (only supported for SQDIFF and CCORR_NORMED, same type and size as ipTemplateImage) *)
		fScaleFactor	:	REAL;	(* Factor (0..1] to reduce source and template image width and height for better performance (but less accuracy!) *)
		eInterpolationType	:	ETcVnInterpolationType;	(* Image resize interpolation type (only used if fScaleFactor != 1, TCVN_IT_BILINEAR recommended for most cases) *)
		ipMatchValues	:	REFERENCE TO ITcVnContainer;	(* Optionally returns the matching values (ContainerType_Vector_REAL, same size and sort order as ipMatches. Set to 0 if not required.) *)
		hrPrev	:	HRESULT;	(* HRESULT indicating the result of previous operations (If SUCCEEDED(hrPrev) equals false, no operation is executed.) *)
	END_VAR

END_FUNCTION

// Functions/Basic Container Operations/F_VN_AppendToContainer/F_VN_AppendToContainer_ITcVnContainer

	{attribute 'TcIecLibraryType'}
	{attribute 'external_name' := 'F_VN_AppendToContainer_ITcVnContainer_GUID_60457B72_8A01_5DC7_6347_92044F23F4B1'}
	(* Append a single element to a container or concatenate containers (if ipElement has the same typeId as ipContainer). *)
	FUNCTION F_VN_AppendToContainer_ITcVnContainer : HRESULT
	VAR_INPUT
		ipElement	:	ITcVnContainer;	(* Single element to append to ipContainer or container with several elements to be concatenated *)
		ipContainer	:	ITcVnContainer;	(* Container to which the element(s) will be appended *)
		hrPrev	:	HRESULT;	(* HRESULT indicating the result of previous operations (If SUCCEEDED(hrPrev) equals false, no operation is executed.) *)
	END_VAR

END_FUNCTION

// Functions/Basic Container Operations/F_VN_AppendToContainer/F_VN_AppendToContainer_ITcVnForwardIterator

	{attribute 'TcIecLibraryType'}
	{attribute 'external_name' := 'F_VN_AppendToContainer_ITcVnForwardIterator_GUID_00CA9150_1665_5F67_4B19_E7594F3029B4'}
	(* Append a single element (represented by an iterator)to a container. *)
	FUNCTION F_VN_AppendToContainer_ITcVnForwardIterator : HRESULT
	VAR_INPUT
		ipElement	:	ITcVnForwardIterator;	(* Single element to append to ipContainer *)
		ipContainer	:	ITcVnContainer;	(* Container to which the element(s) will be appended *)
		hrPrev	:	HRESULT;	(* HRESULT indicating the result of previous operations (If SUCCEEDED(hrPrev) equals false, no operation is executed.) *)
	END_VAR

END_FUNCTION

// Functions/Basic Container Operations/F_VN_AppendToContainer/F_VN_AppendToContainer_DINT

	{attribute 'TcIecLibraryType'}
	{attribute 'external_name' := 'F_VN_AppendToContainer_DINT_GUID_ADD74149_F093_5F6A_52CB_1A431F2060B2'}
	(* Append a single element of type DINT to a container. *)
	FUNCTION F_VN_AppendToContainer_DINT : HRESULT
	VAR_INPUT
		nElement	:	DINT;	(* Single element to append to ipContainer *)
		ipContainer	:	ITcVnContainer;	(* Container to which the element will be appended *)
		hrPrev	:	HRESULT;	(* HRESULT indicating the result of previous operations (If SUCCEEDED(hrPrev) equals false, no operation is executed.) *)
	END_VAR

END_FUNCTION

// Functions/Basic Container Operations/F_VN_AppendToContainer/F_VN_AppendToContainer_LREAL

	{attribute 'TcIecLibraryType'}
	{attribute 'external_name' := 'F_VN_AppendToContainer_LREAL_GUID_5A1A5F61_538E_53B2_674A_9F7A0FB17D88'}
	(* Append a single element of type LREAL to a container. *)
	FUNCTION F_VN_AppendToContainer_LREAL : HRESULT
	VAR_INPUT
		fElement	:	LREAL;	(* Single element to append to ipContainer *)
		ipContainer	:	ITcVnContainer;	(* Container to which the element will be appended *)
		hrPrev	:	HRESULT;	(* HRESULT indicating the result of previous operations (If SUCCEEDED(hrPrev) equals false, no operation is executed.) *)
	END_VAR

END_FUNCTION

// Functions/Basic Container Operations/F_VN_AppendToContainer/F_VN_AppendToContainer_REAL

	{attribute 'TcIecLibraryType'}
	{attribute 'external_name' := 'F_VN_AppendToContainer_REAL_GUID_431F873E_1849_5546_7ECE_5AEA6CFFE222'}
	(* Append a single element of type REAL to a container. *)
	FUNCTION F_VN_AppendToContainer_REAL : HRESULT
	VAR_INPUT
		fElement	:	REAL;	(* Single element to append to ipContainer *)
		ipContainer	:	ITcVnContainer;	(* Container to which the element will be appended *)
		hrPrev	:	HRESULT;	(* HRESULT indicating the result of previous operations (If SUCCEEDED(hrPrev) equals false, no operation is executed.) *)
	END_VAR

END_FUNCTION

// Functions/Basic Container Operations/F_VN_AppendToContainer/F_VN_AppendToContainer_SINT

	{attribute 'TcIecLibraryType'}
	{attribute 'external_name' := 'F_VN_AppendToContainer_SINT_GUID_C53A1634_AAC2_59EC_7A29_3733D2445750'}
	(* Append a single element of type SINT to a container. *)
	FUNCTION F_VN_AppendToContainer_SINT : HRESULT
	VAR_INPUT
		nElement	:	SINT;	(* Single element to append to ipContainer *)
		ipContainer	:	ITcVnContainer;	(* Container to which the element will be appended *)
		hrPrev	:	HRESULT;	(* HRESULT indicating the result of previous operations (If SUCCEEDED(hrPrev) equals false, no operation is executed.) *)
	END_VAR

END_FUNCTION

// Functions/Basic Container Operations/F_VN_AppendToContainer/F_VN_AppendToContainer_TcVnDMatch

	{attribute 'TcIecLibraryType'}
	{attribute 'external_name' := 'F_VN_AppendToContainer_TcVnDMatch_GUID_DF3C224B_EE95_5E63_777A_B55B8E610FAE'}
	(* Append a single element of type TcVnDMatch to a container. *)
	FUNCTION F_VN_AppendToContainer_TcVnDMatch : HRESULT
	VAR_INPUT
		stElement	:	REFERENCE TO TcVnDMatch;	(* Single element to append to ipContainer *)
		ipContainer	:	ITcVnContainer;	(* Container to which the element will be appended *)
		hrPrev	:	HRESULT;	(* HRESULT indicating the result of previous operations (If SUCCEEDED(hrPrev) equals false, no operation is executed.) *)
	END_VAR

END_FUNCTION

// Functions/Basic Container Operations/F_VN_AppendToContainer/F_VN_AppendToContainer_TcVnKeyPoint

	{attribute 'TcIecLibraryType'}
	{attribute 'external_name' := 'F_VN_AppendToContainer_TcVnKeyPoint_GUID_36A421AF_C0A8_5B40_62E9_0F1DEFDCBB42'}
	(* Append a single element of type TcVnKeyPoint to a container. *)
	FUNCTION F_VN_AppendToContainer_TcVnKeyPoint : HRESULT
	VAR_INPUT
		stElement	:	REFERENCE TO TcVnKeyPoint;	(* Single element to append to ipContainer *)
		ipContainer	:	ITcVnContainer;	(* Container to which the element will be appended *)
		hrPrev	:	HRESULT;	(* HRESULT indicating the result of previous operations (If SUCCEEDED(hrPrev) equals false, no operation is executed.) *)
	END_VAR

END_FUNCTION

// Functions/Basic Container Operations/F_VN_AppendToContainer/F_VN_AppendToContainer_TcVnPoint2_DINT

	{attribute 'TcIecLibraryType'}
	{attribute 'external_name' := 'F_VN_AppendToContainer_TcVnPoint2_DINT_GUID_098E9B37_546B_52D6_5026_FA14C0FA7048'}
	(* Append a single element of type TcVnPoint2_DINT to a container. *)
	FUNCTION F_VN_AppendToContainer_TcVnPoint2_DINT : HRESULT
	VAR_INPUT
		aElement	:	REFERENCE TO TcVnPoint2_DINT;	(* Single element to append to ipContainer *)
		ipContainer	:	ITcVnContainer;	(* Container to which the element will be appended *)
		hrPrev	:	HRESULT;	(* HRESULT indicating the result of previous operations (If SUCCEEDED(hrPrev) equals false, no operation is executed.) *)
	END_VAR

END_FUNCTION

// Functions/Basic Container Operations/F_VN_AppendToContainer/F_VN_AppendToContainer_TcVnPoint2_LREAL

	{attribute 'TcIecLibraryType'}
	{attribute 'external_name' := 'F_VN_AppendToContainer_TcVnPoint2_LREAL_GUID_FD4C7911_2FC5_5B00_48BD_2CAFB58E5B83'}
	(* Append a single element of type TcVnPoint2_LREAL to a container. *)
	FUNCTION F_VN_AppendToContainer_TcVnPoint2_LREAL : HRESULT
	VAR_INPUT
		aElement	:	REFERENCE TO TcVnPoint2_LREAL;	(* Single element to append to ipContainer *)
		ipContainer	:	ITcVnContainer;	(* Container to which the element will be appended *)
		hrPrev	:	HRESULT;	(* HRESULT indicating the result of previous operations (If SUCCEEDED(hrPrev) equals false, no operation is executed.) *)
	END_VAR

END_FUNCTION

// Functions/Basic Container Operations/F_VN_AppendToContainer/F_VN_AppendToContainer_TcVnPoint2_REAL

	{attribute 'TcIecLibraryType'}
	{attribute 'external_name' := 'F_VN_AppendToContainer_TcVnPoint2_REAL_GUID_449819B3_535C_5F4E_63CB_8A7B99BD5BC9'}
	(* Append a single element of type TcVnPoint2_REAL to a container. *)
	FUNCTION F_VN_AppendToContainer_TcVnPoint2_REAL : HRESULT
	VAR_INPUT
		aElement	:	REFERENCE TO TcVnPoint2_REAL;	(* Single element to append to ipContainer *)
		ipContainer	:	ITcVnContainer;	(* Container to which the element will be appended *)
		hrPrev	:	HRESULT;	(* HRESULT indicating the result of previous operations (If SUCCEEDED(hrPrev) equals false, no operation is executed.) *)
	END_VAR

END_FUNCTION

// Functions/Basic Container Operations/F_VN_AppendToContainer/F_VN_AppendToContainer_TcVnPoint3_LREAL

	{attribute 'TcIecLibraryType'}
	{attribute 'external_name' := 'F_VN_AppendToContainer_TcVnPoint3_LREAL_GUID_A83918A9_A33D_5C71_4233_83D99A8EF2E7'}
	(* Append a single element of type TcVnPoint3_LREAL to a container. *)
	FUNCTION F_VN_AppendToContainer_TcVnPoint3_LREAL : HRESULT
	VAR_INPUT
		aElement	:	REFERENCE TO TcVnPoint3_LREAL;	(* Single element to append to ipContainer *)
		ipContainer	:	ITcVnContainer;	(* Container to which the element will be appended *)
		hrPrev	:	HRESULT;	(* HRESULT indicating the result of previous operations (If SUCCEEDED(hrPrev) equals false, no operation is executed.) *)
	END_VAR

END_FUNCTION

// Functions/Basic Container Operations/F_VN_AppendToContainer/F_VN_AppendToContainer_TcVnPoint3_REAL

	{attribute 'TcIecLibraryType'}
	{attribute 'external_name' := 'F_VN_AppendToContainer_TcVnPoint3_REAL_GUID_B4E18A9D_E30C_5BCF_5EE3_C498E1D371D0'}
	(* Append a single element of type TcVnPoint3_REAL to a container. *)
	FUNCTION F_VN_AppendToContainer_TcVnPoint3_REAL : HRESULT
	VAR_INPUT
		aElement	:	REFERENCE TO TcVnPoint3_REAL;	(* Single element to append to ipContainer *)
		ipContainer	:	ITcVnContainer;	(* Container to which the element will be appended *)
		hrPrev	:	HRESULT;	(* HRESULT indicating the result of previous operations (If SUCCEEDED(hrPrev) equals false, no operation is executed.) *)
	END_VAR

END_FUNCTION

// Functions/Basic Container Operations/F_VN_AppendToContainer/F_VN_AppendToContainer_TcVnRectangle_DINT

	{attribute 'TcIecLibraryType'}
	{attribute 'external_name' := 'F_VN_AppendToContainer_TcVnRectangle_DINT_GUID_AC9CAD73_CCCA_598D_4863_D986C9280D73'}
	(* Append a single element of type TcVnRectangle_DINT to a container. *)
	FUNCTION F_VN_AppendToContainer_TcVnRectangle_DINT : HRESULT
	VAR_INPUT
		stElement	:	REFERENCE TO TcVnRectangle_DINT;	(* Single element to append to ipContainer *)
		ipContainer	:	ITcVnContainer;	(* Container to which the element will be appended *)
		hrPrev	:	HRESULT;	(* HRESULT indicating the result of previous operations (If SUCCEEDED(hrPrev) equals false, no operation is executed.) *)
	END_VAR

END_FUNCTION

// Functions/Basic Container Operations/F_VN_AppendToContainer/F_VN_AppendToContainer_TcVnVector2_DINT

	{attribute 'TcIecLibraryType'}
	{attribute 'external_name' := 'F_VN_AppendToContainer_TcVnVector2_DINT_GUID_2987FBBD_4AF0_580F_7DA0_581EBDFBFB58'}
	(* Append a single element of type TcVnVector2_DINT to a container. *)
	FUNCTION F_VN_AppendToContainer_TcVnVector2_DINT : HRESULT
	VAR_INPUT
		aElement	:	REFERENCE TO TcVnVector2_DINT;	(* Single element to append to ipContainer *)
		ipContainer	:	ITcVnContainer;	(* Container to which the element will be appended *)
		hrPrev	:	HRESULT;	(* HRESULT indicating the result of previous operations (If SUCCEEDED(hrPrev) equals false, no operation is executed.) *)
	END_VAR

END_FUNCTION

// Functions/Basic Container Operations/F_VN_AppendToContainer/F_VN_AppendToContainer_TcVnVector2_REAL

	{attribute 'TcIecLibraryType'}
	{attribute 'external_name' := 'F_VN_AppendToContainer_TcVnVector2_REAL_GUID_A29DA2E3_3956_599D_63A3_465B51E93854'}
	(* Append a single element of type TcVnVector2_REAL to a container. *)
	FUNCTION F_VN_AppendToContainer_TcVnVector2_REAL : HRESULT
	VAR_INPUT
		aElement	:	REFERENCE TO TcVnVector2_REAL;	(* Single element to append to ipContainer *)
		ipContainer	:	ITcVnContainer;	(* Container to which the element will be appended *)
		hrPrev	:	HRESULT;	(* HRESULT indicating the result of previous operations (If SUCCEEDED(hrPrev) equals false, no operation is executed.) *)
	END_VAR

END_FUNCTION

// Functions/Basic Container Operations/F_VN_AppendToContainer/F_VN_AppendToContainer_TcVnVector3_REAL

	{attribute 'TcIecLibraryType'}
	{attribute 'external_name' := 'F_VN_AppendToContainer_TcVnVector3_REAL_GUID_BAF84BA3_B50A_5FB3_53DB_6493EB8FA2D2'}
	(* Append a single element of type TcVnVector3_REAL to a container. *)
	FUNCTION F_VN_AppendToContainer_TcVnVector3_REAL : HRESULT
	VAR_INPUT
		aElement	:	REFERENCE TO TcVnVector3_REAL;	(* Single element to append to ipContainer *)
		ipContainer	:	ITcVnContainer;	(* Container to which the element will be appended *)
		hrPrev	:	HRESULT;	(* HRESULT indicating the result of previous operations (If SUCCEEDED(hrPrev) equals false, no operation is executed.) *)
	END_VAR

END_FUNCTION

// Functions/Basic Container Operations/F_VN_AppendToContainer/F_VN_AppendToContainer_TcVnVector4_DINT

	{attribute 'TcIecLibraryType'}
	{attribute 'external_name' := 'F_VN_AppendToContainer_TcVnVector4_DINT_GUID_E3875633_C399_5105_780B_E8FA5DAB4D3D'}
	(* Append a single element of type TcVnVector4_DINT to a container. *)
	FUNCTION F_VN_AppendToContainer_TcVnVector4_DINT : HRESULT
	VAR_INPUT
		aElement	:	REFERENCE TO TcVnVector4_DINT;	(* Single element to append to ipContainer *)
		ipContainer	:	ITcVnContainer;	(* Container to which the element will be appended *)
		hrPrev	:	HRESULT;	(* HRESULT indicating the result of previous operations (If SUCCEEDED(hrPrev) equals false, no operation is executed.) *)
	END_VAR

END_FUNCTION

// Functions/Basic Container Operations/F_VN_AppendToContainer/F_VN_AppendToContainer_TcVnVector4_LREAL

	{attribute 'TcIecLibraryType'}
	{attribute 'external_name' := 'F_VN_AppendToContainer_TcVnVector4_LREAL_GUID_83A5882E_3644_570D_7415_0DF0B60E1AFF'}
	(* Append a single element of type TcVnVector4_LREAL to a container. *)
	FUNCTION F_VN_AppendToContainer_TcVnVector4_LREAL : HRESULT
	VAR_INPUT
		aElement	:	REFERENCE TO TcVnVector4_LREAL;	(* Single element to append to ipContainer *)
		ipContainer	:	ITcVnContainer;	(* Container to which the element will be appended *)
		hrPrev	:	HRESULT;	(* HRESULT indicating the result of previous operations (If SUCCEEDED(hrPrev) equals false, no operation is executed.) *)
	END_VAR

END_FUNCTION

// Functions/Basic Container Operations/F_VN_AppendToContainer/F_VN_AppendToContainer_UDINT

	{attribute 'TcIecLibraryType'}
	{attribute 'external_name' := 'F_VN_AppendToContainer_UDINT_GUID_6FC8A047_231F_5DD3_4423_E6D4D3B7D883'}
	(* Append a single element of type UDINT to a container. *)
	FUNCTION F_VN_AppendToContainer_UDINT : HRESULT
	VAR_INPUT
		nElement	:	UDINT;	(* Single element to append to ipContainer *)
		ipContainer	:	ITcVnContainer;	(* Container to which the element will be appended *)
		hrPrev	:	HRESULT;	(* HRESULT indicating the result of previous operations (If SUCCEEDED(hrPrev) equals false, no operation is executed.) *)
	END_VAR

END_FUNCTION

// Functions/Basic Container Operations/F_VN_AppendToContainer/F_VN_AppendToContainer_ULINT

	{attribute 'TcIecLibraryType'}
	{attribute 'external_name' := 'F_VN_AppendToContainer_ULINT_GUID_599EFC7C_4409_597D_71AE_EB0193F6DBDE'}
	(* Append a single element of type ULINT to a container. *)
	FUNCTION F_VN_AppendToContainer_ULINT : HRESULT
	VAR_INPUT
		nElement	:	ULINT;	(* Single element to append to ipContainer *)
		ipContainer	:	ITcVnContainer;	(* Container to which the element will be appended *)
		hrPrev	:	HRESULT;	(* HRESULT indicating the result of previous operations (If SUCCEEDED(hrPrev) equals false, no operation is executed.) *)
	END_VAR

END_FUNCTION

// Functions/Basic Container Operations/F_VN_FillContainer/F_VN_FillContainer_DINT

	{attribute 'TcIecLibraryType'}
	{attribute 'external_name' := 'F_VN_FillContainer_DINT_GUID_E386D310_7104_5B51_6577_FFAE22583F85'}
	(* Fill the container with the specified value. Only possible for containers with basic elements. *)
	FUNCTION F_VN_FillContainer_DINT : HRESULT
	VAR_INPUT
		ipContainer	:	ITcVnContainer;	(* Container with basic elements *)
		nValue	:	DINT;	(* Value to set the container elements *)
		hrPrev	:	HRESULT;	(* HRESULT indicating the result of previous operations (If SUCCEEDED(hrPrev) equals false, no operation is executed.) *)
	END_VAR

END_FUNCTION

// Functions/Basic Container Operations/F_VN_FillContainer/F_VN_FillContainer_LREAL

	{attribute 'TcIecLibraryType'}
	{attribute 'external_name' := 'F_VN_FillContainer_LREAL_GUID_66874FD1_8799_548F_64D4_8224E2AED892'}
	(* Fill the container with the specified value. Only possible for containers with basic elements. *)
	FUNCTION F_VN_FillContainer_LREAL : HRESULT
	VAR_INPUT
		ipContainer	:	ITcVnContainer;	(* Container with basic elements *)
		fValue	:	LREAL;	(* Value to set the container elements *)
		hrPrev	:	HRESULT;	(* HRESULT indicating the result of previous operations (If SUCCEEDED(hrPrev) equals false, no operation is executed.) *)
	END_VAR

END_FUNCTION

// Functions/Basic Container Operations/F_VN_FillContainer/F_VN_FillContainer_REAL

	{attribute 'TcIecLibraryType'}
	{attribute 'external_name' := 'F_VN_FillContainer_REAL_GUID_3B8D6183_9EBE_5E56_5A6C_1145416411A8'}
	(* Fill the container with the specified value. Only possible for containers with basic elements. *)
	FUNCTION F_VN_FillContainer_REAL : HRESULT
	VAR_INPUT
		ipContainer	:	ITcVnContainer;	(* Container with basic elements *)
		fValue	:	REAL;	(* Value to set the container elements *)
		hrPrev	:	HRESULT;	(* HRESULT indicating the result of previous operations (If SUCCEEDED(hrPrev) equals false, no operation is executed.) *)
	END_VAR

END_FUNCTION

// Functions/Basic Container Operations/F_VN_FillContainer/F_VN_FillContainer_SINT

	{attribute 'TcIecLibraryType'}
	{attribute 'external_name' := 'F_VN_FillContainer_SINT_GUID_1CB12694_E95D_5C72_68E3_22FA232EEB9D'}
	(* Fill the container with the specified value. Only possible for containers with basic elements. *)
	FUNCTION F_VN_FillContainer_SINT : HRESULT
	VAR_INPUT
		ipContainer	:	ITcVnContainer;	(* Container with basic elements *)
		nValue	:	SINT;	(* Value to set the container elements *)
		hrPrev	:	HRESULT;	(* HRESULT indicating the result of previous operations (If SUCCEEDED(hrPrev) equals false, no operation is executed.) *)
	END_VAR

END_FUNCTION

// Functions/Basic Container Operations/F_VN_FillContainer/F_VN_FillContainer_TcVnDMatch

	{attribute 'TcIecLibraryType'}
	{attribute 'external_name' := 'F_VN_FillContainer_TcVnDMatch_GUID_717192A6_965E_5824_6FC6_E33B1E529955'}
	(* Fill the container with the specified value. Only possible for containers with basic elements. *)
	FUNCTION F_VN_FillContainer_TcVnDMatch : HRESULT
	VAR_INPUT
		ipContainer	:	ITcVnContainer;	(* Container with basic elements *)
		stValue	:	REFERENCE TO TcVnDMatch;	(* Value to set the container elements *)
		hrPrev	:	HRESULT;	(* HRESULT indicating the result of previous operations (If SUCCEEDED(hrPrev) equals false, no operation is executed.) *)
	END_VAR

END_FUNCTION

// Functions/Basic Container Operations/F_VN_FillContainer/F_VN_FillContainer_TcVnKeyPoint

	{attribute 'TcIecLibraryType'}
	{attribute 'external_name' := 'F_VN_FillContainer_TcVnKeyPoint_GUID_FBC1DCB2_E8D1_5D77_6627_88840DC4C142'}
	(* Fill the container with the specified value. Only possible for containers with basic elements. *)
	FUNCTION F_VN_FillContainer_TcVnKeyPoint : HRESULT
	VAR_INPUT
		ipContainer	:	ITcVnContainer;	(* Container with basic elements *)
		stValue	:	REFERENCE TO TcVnKeyPoint;	(* Value to set the container elements *)
		hrPrev	:	HRESULT;	(* HRESULT indicating the result of previous operations (If SUCCEEDED(hrPrev) equals false, no operation is executed.) *)
	END_VAR

END_FUNCTION

// Functions/Basic Container Operations/F_VN_FillContainer/F_VN_FillContainer_TcVnPoint2_DINT

	{attribute 'TcIecLibraryType'}
	{attribute 'external_name' := 'F_VN_FillContainer_TcVnPoint2_DINT_GUID_E15E13EE_14CA_5507_69EA_2AA6C84AAEA3'}
	(* Fill the container with the specified value. Only possible for containers with basic elements. *)
	FUNCTION F_VN_FillContainer_TcVnPoint2_DINT : HRESULT
	VAR_INPUT
		ipContainer	:	ITcVnContainer;	(* Container with basic elements *)
		aValue	:	REFERENCE TO TcVnPoint2_DINT;	(* Value to set the container elements *)
		hrPrev	:	HRESULT;	(* HRESULT indicating the result of previous operations (If SUCCEEDED(hrPrev) equals false, no operation is executed.) *)
	END_VAR

END_FUNCTION

// Functions/Basic Container Operations/F_VN_FillContainer/F_VN_FillContainer_TcVnPoint2_LREAL

	{attribute 'TcIecLibraryType'}
	{attribute 'external_name' := 'F_VN_FillContainer_TcVnPoint2_LREAL_GUID_4183E683_CADE_536B_405C_F1F3CF0F0661'}
	(* Fill the container with the specified value. Only possible for containers with basic elements. *)
	FUNCTION F_VN_FillContainer_TcVnPoint2_LREAL : HRESULT
	VAR_INPUT
		ipContainer	:	ITcVnContainer;	(* Container with basic elements *)
		aValue	:	REFERENCE TO TcVnPoint2_LREAL;	(* Value to set the container elements *)
		hrPrev	:	HRESULT;	(* HRESULT indicating the result of previous operations (If SUCCEEDED(hrPrev) equals false, no operation is executed.) *)
	END_VAR

END_FUNCTION

// Functions/Basic Container Operations/F_VN_FillContainer/F_VN_FillContainer_TcVnPoint2_REAL

	{attribute 'TcIecLibraryType'}
	{attribute 'external_name' := 'F_VN_FillContainer_TcVnPoint2_REAL_GUID_EE325A29_14E9_59A9_6FB8_9A708073E152'}
	(* Fill the container with the specified value. Only possible for containers with basic elements. *)
	FUNCTION F_VN_FillContainer_TcVnPoint2_REAL : HRESULT
	VAR_INPUT
		ipContainer	:	ITcVnContainer;	(* Container with basic elements *)
		aValue	:	REFERENCE TO TcVnPoint2_REAL;	(* Value to set the container elements *)
		hrPrev	:	HRESULT;	(* HRESULT indicating the result of previous operations (If SUCCEEDED(hrPrev) equals false, no operation is executed.) *)
	END_VAR

END_FUNCTION

// Functions/Basic Container Operations/F_VN_FillContainer/F_VN_FillContainer_TcVnPoint3_LREAL

	{attribute 'TcIecLibraryType'}
	{attribute 'external_name' := 'F_VN_FillContainer_TcVnPoint3_LREAL_GUID_15721FBE_13AC_5DDC_596B_BF11259626E4'}
	(* Fill the container with the specified value. Only possible for containers with basic elements. *)
	FUNCTION F_VN_FillContainer_TcVnPoint3_LREAL : HRESULT
	VAR_INPUT
		ipContainer	:	ITcVnContainer;	(* Container with basic elements *)
		aValue	:	REFERENCE TO TcVnPoint3_LREAL;	(* Value to set the container elements *)
		hrPrev	:	HRESULT;	(* HRESULT indicating the result of previous operations (If SUCCEEDED(hrPrev) equals false, no operation is executed.) *)
	END_VAR

END_FUNCTION

// Functions/Basic Container Operations/F_VN_FillContainer/F_VN_FillContainer_TcVnPoint3_REAL

	{attribute 'TcIecLibraryType'}
	{attribute 'external_name' := 'F_VN_FillContainer_TcVnPoint3_REAL_GUID_F4FBFCCD_7C13_5C66_63C5_A63782E5ABA7'}
	(* Fill the container with the specified value. Only possible for containers with basic elements. *)
	FUNCTION F_VN_FillContainer_TcVnPoint3_REAL : HRESULT
	VAR_INPUT
		ipContainer	:	ITcVnContainer;	(* Container with basic elements *)
		aValue	:	REFERENCE TO TcVnPoint3_REAL;	(* Value to set the container elements *)
		hrPrev	:	HRESULT;	(* HRESULT indicating the result of previous operations (If SUCCEEDED(hrPrev) equals false, no operation is executed.) *)
	END_VAR

END_FUNCTION

// Functions/Basic Container Operations/F_VN_FillContainer/F_VN_FillContainer_TcVnRectangle_DINT

	{attribute 'TcIecLibraryType'}
	{attribute 'external_name' := 'F_VN_FillContainer_TcVnRectangle_DINT_GUID_8432DF21_3564_5097_47DA_81185018ED41'}
	(* Fill the container with the specified value. Only possible for containers with basic elements. *)
	FUNCTION F_VN_FillContainer_TcVnRectangle_DINT : HRESULT
	VAR_INPUT
		ipContainer	:	ITcVnContainer;	(* Container with basic elements *)
		stValue	:	REFERENCE TO TcVnRectangle_DINT;	(* Value to set the container elements *)
		hrPrev	:	HRESULT;	(* HRESULT indicating the result of previous operations (If SUCCEEDED(hrPrev) equals false, no operation is executed.) *)
	END_VAR

END_FUNCTION

// Functions/Basic Container Operations/F_VN_FillContainer/F_VN_FillContainer_TcVnVector2_DINT

	{attribute 'TcIecLibraryType'}
	{attribute 'external_name' := 'F_VN_FillContainer_TcVnVector2_DINT_GUID_BEA6D692_99BF_5AED_40E2_E555455971FA'}
	(* Fill the container with the specified value. Only possible for containers with basic elements. *)
	FUNCTION F_VN_FillContainer_TcVnVector2_DINT : HRESULT
	VAR_INPUT
		ipContainer	:	ITcVnContainer;	(* Container with basic elements *)
		aValue	:	REFERENCE TO TcVnVector2_DINT;	(* Value to set the container elements *)
		hrPrev	:	HRESULT;	(* HRESULT indicating the result of previous operations (If SUCCEEDED(hrPrev) equals false, no operation is executed.) *)
	END_VAR

END_FUNCTION

// Functions/Basic Container Operations/F_VN_FillContainer/F_VN_FillContainer_TcVnVector2_REAL

	{attribute 'TcIecLibraryType'}
	{attribute 'external_name' := 'F_VN_FillContainer_TcVnVector2_REAL_GUID_2967B180_87F1_5452_73E8_1A0D4A357B9E'}
	(* Fill the container with the specified value. Only possible for containers with basic elements. *)
	FUNCTION F_VN_FillContainer_TcVnVector2_REAL : HRESULT
	VAR_INPUT
		ipContainer	:	ITcVnContainer;	(* Container with basic elements *)
		aValue	:	REFERENCE TO TcVnVector2_REAL;	(* Value to set the container elements *)
		hrPrev	:	HRESULT;	(* HRESULT indicating the result of previous operations (If SUCCEEDED(hrPrev) equals false, no operation is executed.) *)
	END_VAR

END_FUNCTION

// Functions/Basic Container Operations/F_VN_FillContainer/F_VN_FillContainer_TcVnVector3_REAL

	{attribute 'TcIecLibraryType'}
	{attribute 'external_name' := 'F_VN_FillContainer_TcVnVector3_REAL_GUID_7081F4D4_F32D_5DA4_4D11_B7DC87C60028'}
	(* Fill the container with the specified value. Only possible for containers with basic elements. *)
	FUNCTION F_VN_FillContainer_TcVnVector3_REAL : HRESULT
	VAR_INPUT
		ipContainer	:	ITcVnContainer;	(* Container with basic elements *)
		aValue	:	REFERENCE TO TcVnVector3_REAL;	(* Value to set the container elements *)
		hrPrev	:	HRESULT;	(* HRESULT indicating the result of previous operations (If SUCCEEDED(hrPrev) equals false, no operation is executed.) *)
	END_VAR

END_FUNCTION

// Functions/Basic Container Operations/F_VN_FillContainer/F_VN_FillContainer_TcVnVector4_DINT

	{attribute 'TcIecLibraryType'}
	{attribute 'external_name' := 'F_VN_FillContainer_TcVnVector4_DINT_GUID_7FA061F7_4EF8_5A84_6B43_85A73AB1C0C7'}
	(* Fill the container with the specified value. Only possible for containers with basic elements. *)
	FUNCTION F_VN_FillContainer_TcVnVector4_DINT : HRESULT
	VAR_INPUT
		ipContainer	:	ITcVnContainer;	(* Container with basic elements *)
		aValue	:	REFERENCE TO TcVnVector4_DINT;	(* Value to set the container elements *)
		hrPrev	:	HRESULT;	(* HRESULT indicating the result of previous operations (If SUCCEEDED(hrPrev) equals false, no operation is executed.) *)
	END_VAR

END_FUNCTION

// Functions/Basic Container Operations/F_VN_FillContainer/F_VN_FillContainer_TcVnVector4_LREAL

	{attribute 'TcIecLibraryType'}
	{attribute 'external_name' := 'F_VN_FillContainer_TcVnVector4_LREAL_GUID_A620FB05_EB97_53BF_588E_DF79BF9834A3'}
	(* Fill the container with the specified value. Only possible for containers with basic elements. *)
	FUNCTION F_VN_FillContainer_TcVnVector4_LREAL : HRESULT
	VAR_INPUT
		ipContainer	:	ITcVnContainer;	(* Container with basic elements *)
		aValue	:	REFERENCE TO TcVnVector4_LREAL;	(* Value to set the container elements *)
		hrPrev	:	HRESULT;	(* HRESULT indicating the result of previous operations (If SUCCEEDED(hrPrev) equals false, no operation is executed.) *)
	END_VAR

END_FUNCTION

// Functions/Basic Container Operations/F_VN_FillContainer/F_VN_FillContainer_UDINT

	{attribute 'TcIecLibraryType'}
	{attribute 'external_name' := 'F_VN_FillContainer_UDINT_GUID_C82F2CA8_4257_5A1F_41A3_2EC0D7C00802'}
	(* Fill the container with the specified value. Only possible for containers with basic elements. *)
	FUNCTION F_VN_FillContainer_UDINT : HRESULT
	VAR_INPUT
		ipContainer	:	ITcVnContainer;	(* Container with basic elements *)
		nValue	:	UDINT;	(* Value to set the container elements *)
		hrPrev	:	HRESULT;	(* HRESULT indicating the result of previous operations (If SUCCEEDED(hrPrev) equals false, no operation is executed.) *)
	END_VAR

END_FUNCTION

// Functions/Basic Container Operations/F_VN_FillContainer/F_VN_FillContainer_ULINT

	{attribute 'TcIecLibraryType'}
	{attribute 'external_name' := 'F_VN_FillContainer_ULINT_GUID_F5A7BA95_9E94_59FE_6534_081DA457A462'}
	(* Fill the container with the specified value. Only possible for containers with basic elements. *)
	FUNCTION F_VN_FillContainer_ULINT : HRESULT
	VAR_INPUT
		ipContainer	:	ITcVnContainer;	(* Container with basic elements *)
		nValue	:	ULINT;	(* Value to set the container elements *)
		hrPrev	:	HRESULT;	(* HRESULT indicating the result of previous operations (If SUCCEEDED(hrPrev) equals false, no operation is executed.) *)
	END_VAR

END_FUNCTION

// Functions/Basic Container Operations/F_VN_FillContainerExp/F_VN_FillContainerExp_DINT

	{attribute 'TcIecLibraryType'}
	{attribute 'external_name' := 'F_VN_FillContainerExp_DINT_GUID_24C2AC73_8969_5B85_6A69_88BD02EF2F78'}
	(* Partially fill the container with the specified value. Only possible for containers with basic elements. (expert function) *)
	FUNCTION F_VN_FillContainerExp_DINT : HRESULT
	VAR_INPUT
		ipContainer	:	ITcVnContainer;	(* Container with basic elements *)
		nValue	:	DINT;	(* Value to set the container elements *)
		nStartIdx	:	ULINT;	(* Start index *)
		nCount	:	ULINT;	(* Number of elements to set *)
		hrPrev	:	HRESULT;	(* HRESULT indicating the result of previous operations (If SUCCEEDED(hrPrev) equals false, no operation is executed.) *)
	END_VAR

END_FUNCTION

// Functions/Basic Container Operations/F_VN_FillContainerExp/F_VN_FillContainerExp_LREAL

	{attribute 'TcIecLibraryType'}
	{attribute 'external_name' := 'F_VN_FillContainerExp_LREAL_GUID_9ABD388E_9685_556C_6267_78B2D7AF9DBE'}
	(* Partially fill the container with the specified value. Only possible for containers with basic elements. (expert function) *)
	FUNCTION F_VN_FillContainerExp_LREAL : HRESULT
	VAR_INPUT
		ipContainer	:	ITcVnContainer;	(* Container with basic elements *)
		fValue	:	LREAL;	(* Value to set the container elements *)
		nStartIdx	:	ULINT;	(* Start index *)
		nCount	:	ULINT;	(* Number of elements to set *)
		hrPrev	:	HRESULT;	(* HRESULT indicating the result of previous operations (If SUCCEEDED(hrPrev) equals false, no operation is executed.) *)
	END_VAR

END_FUNCTION

// Functions/Basic Container Operations/F_VN_FillContainerExp/F_VN_FillContainerExp_REAL

	{attribute 'TcIecLibraryType'}
	{attribute 'external_name' := 'F_VN_FillContainerExp_REAL_GUID_D4AD8B99_8C51_56A6_52A2_EF4C6D2BE46D'}
	(* Partially fill the container with the specified value. Only possible for containers with basic elements. (expert function) *)
	FUNCTION F_VN_FillContainerExp_REAL : HRESULT
	VAR_INPUT
		ipContainer	:	ITcVnContainer;	(* Container with basic elements *)
		fValue	:	REAL;	(* Value to set the container elements *)
		nStartIdx	:	ULINT;	(* Start index *)
		nCount	:	ULINT;	(* Number of elements to set *)
		hrPrev	:	HRESULT;	(* HRESULT indicating the result of previous operations (If SUCCEEDED(hrPrev) equals false, no operation is executed.) *)
	END_VAR

END_FUNCTION

// Functions/Basic Container Operations/F_VN_FillContainerExp/F_VN_FillContainerExp_SINT

	{attribute 'TcIecLibraryType'}
	{attribute 'external_name' := 'F_VN_FillContainerExp_SINT_GUID_0C93F192_0B07_5BAA_5856_58505CFC6009'}
	(* Partially fill the container with the specified value. Only possible for containers with basic elements. (expert function) *)
	FUNCTION F_VN_FillContainerExp_SINT : HRESULT
	VAR_INPUT
		ipContainer	:	ITcVnContainer;	(* Container with basic elements *)
		nValue	:	SINT;	(* Value to set the container elements *)
		nStartIdx	:	ULINT;	(* Start index *)
		nCount	:	ULINT;	(* Number of elements to set *)
		hrPrev	:	HRESULT;	(* HRESULT indicating the result of previous operations (If SUCCEEDED(hrPrev) equals false, no operation is executed.) *)
	END_VAR

END_FUNCTION

// Functions/Basic Container Operations/F_VN_FillContainerExp/F_VN_FillContainerExp_TcVnDMatch

	{attribute 'TcIecLibraryType'}
	{attribute 'external_name' := 'F_VN_FillContainerExp_TcVnDMatch_GUID_F2A6E472_836F_5B2B_4F73_82E2C1CCDFBB'}
	(* Partially fill the container with the specified value. Only possible for containers with basic elements. (expert function) *)
	FUNCTION F_VN_FillContainerExp_TcVnDMatch : HRESULT
	VAR_INPUT
		ipContainer	:	ITcVnContainer;	(* Container with basic elements *)
		stValue	:	REFERENCE TO TcVnDMatch;	(* Value to set the container elements *)
		nStartIdx	:	ULINT;	(* Start index *)
		nCount	:	ULINT;	(* Number of elements to set *)
		hrPrev	:	HRESULT;	(* HRESULT indicating the result of previous operations (If SUCCEEDED(hrPrev) equals false, no operation is executed.) *)
	END_VAR

END_FUNCTION

// Functions/Basic Container Operations/F_VN_FillContainerExp/F_VN_FillContainerExp_TcVnKeyPoint

	{attribute 'TcIecLibraryType'}
	{attribute 'external_name' := 'F_VN_FillContainerExp_TcVnKeyPoint_GUID_C29929CD_955A_571C_6B10_E481C8BC7856'}
	(* Partially fill the container with the specified value. Only possible for containers with basic elements. (expert function) *)
	FUNCTION F_VN_FillContainerExp_TcVnKeyPoint : HRESULT
	VAR_INPUT
		ipContainer	:	ITcVnContainer;	(* Container with basic elements *)
		stValue	:	REFERENCE TO TcVnKeyPoint;	(* Value to set the container elements *)
		nStartIdx	:	ULINT;	(* Start index *)
		nCount	:	ULINT;	(* Number of elements to set *)
		hrPrev	:	HRESULT;	(* HRESULT indicating the result of previous operations (If SUCCEEDED(hrPrev) equals false, no operation is executed.) *)
	END_VAR

END_FUNCTION

// Functions/Basic Container Operations/F_VN_FillContainerExp/F_VN_FillContainerExp_TcVnPoint2_DINT

	{attribute 'TcIecLibraryType'}
	{attribute 'external_name' := 'F_VN_FillContainerExp_TcVnPoint2_DINT_GUID_C9EC4EC8_AD4A_5B6E_759A_7CB5DD6408B6'}
	(* Partially fill the container with the specified value. Only possible for containers with basic elements. (expert function) *)
	FUNCTION F_VN_FillContainerExp_TcVnPoint2_DINT : HRESULT
	VAR_INPUT
		ipContainer	:	ITcVnContainer;	(* Container with basic elements *)
		aValue	:	REFERENCE TO TcVnPoint2_DINT;	(* Value to set the container elements *)
		nStartIdx	:	ULINT;	(* Start index *)
		nCount	:	ULINT;	(* Number of elements to set *)
		hrPrev	:	HRESULT;	(* HRESULT indicating the result of previous operations (If SUCCEEDED(hrPrev) equals false, no operation is executed.) *)
	END_VAR

END_FUNCTION

// Functions/Basic Container Operations/F_VN_FillContainerExp/F_VN_FillContainerExp_TcVnPoint2_LREAL

	{attribute 'TcIecLibraryType'}
	{attribute 'external_name' := 'F_VN_FillContainerExp_TcVnPoint2_LREAL_GUID_73E47DA4_4A98_5DBA_4B4E_CDC94EDA5FA5'}
	(* Partially fill the container with the specified value. Only possible for containers with basic elements. (expert function) *)
	FUNCTION F_VN_FillContainerExp_TcVnPoint2_LREAL : HRESULT
	VAR_INPUT
		ipContainer	:	ITcVnContainer;	(* Container with basic elements *)
		aValue	:	REFERENCE TO TcVnPoint2_LREAL;	(* Value to set the container elements *)
		nStartIdx	:	ULINT;	(* Start index *)
		nCount	:	ULINT;	(* Number of elements to set *)
		hrPrev	:	HRESULT;	(* HRESULT indicating the result of previous operations (If SUCCEEDED(hrPrev) equals false, no operation is executed.) *)
	END_VAR

END_FUNCTION

// Functions/Basic Container Operations/F_VN_FillContainerExp/F_VN_FillContainerExp_TcVnPoint2_REAL

	{attribute 'TcIecLibraryType'}
	{attribute 'external_name' := 'F_VN_FillContainerExp_TcVnPoint2_REAL_GUID_4E80DF29_9041_584F_4166_0847769B775E'}
	(* Partially fill the container with the specified value. Only possible for containers with basic elements. (expert function) *)
	FUNCTION F_VN_FillContainerExp_TcVnPoint2_REAL : HRESULT
	VAR_INPUT
		ipContainer	:	ITcVnContainer;	(* Container with basic elements *)
		aValue	:	REFERENCE TO TcVnPoint2_REAL;	(* Value to set the container elements *)
		nStartIdx	:	ULINT;	(* Start index *)
		nCount	:	ULINT;	(* Number of elements to set *)
		hrPrev	:	HRESULT;	(* HRESULT indicating the result of previous operations (If SUCCEEDED(hrPrev) equals false, no operation is executed.) *)
	END_VAR

END_FUNCTION

// Functions/Basic Container Operations/F_VN_FillContainerExp/F_VN_FillContainerExp_TcVnPoint3_LREAL

	{attribute 'TcIecLibraryType'}
	{attribute 'external_name' := 'F_VN_FillContainerExp_TcVnPoint3_LREAL_GUID_2B7D7CC4_E632_5E6B_5581_75895AA5675B'}
	(* Partially fill the container with the specified value. Only possible for containers with basic elements. (expert function) *)
	FUNCTION F_VN_FillContainerExp_TcVnPoint3_LREAL : HRESULT
	VAR_INPUT
		ipContainer	:	ITcVnContainer;	(* Container with basic elements *)
		aValue	:	REFERENCE TO TcVnPoint3_LREAL;	(* Value to set the container elements *)
		nStartIdx	:	ULINT;	(* Start index *)
		nCount	:	ULINT;	(* Number of elements to set *)
		hrPrev	:	HRESULT;	(* HRESULT indicating the result of previous operations (If SUCCEEDED(hrPrev) equals false, no operation is executed.) *)
	END_VAR

END_FUNCTION

// Functions/Basic Container Operations/F_VN_FillContainerExp/F_VN_FillContainerExp_TcVnPoint3_REAL

	{attribute 'TcIecLibraryType'}
	{attribute 'external_name' := 'F_VN_FillContainerExp_TcVnPoint3_REAL_GUID_F6C1072C_27ED_5E55_5C76_589CF1F3C59D'}
	(* Partially fill the container with the specified value. Only possible for containers with basic elements. (expert function) *)
	FUNCTION F_VN_FillContainerExp_TcVnPoint3_REAL : HRESULT
	VAR_INPUT
		ipContainer	:	ITcVnContainer;	(* Container with basic elements *)
		aValue	:	REFERENCE TO TcVnPoint3_REAL;	(* Value to set the container elements *)
		nStartIdx	:	ULINT;	(* Start index *)
		nCount	:	ULINT;	(* Number of elements to set *)
		hrPrev	:	HRESULT;	(* HRESULT indicating the result of previous operations (If SUCCEEDED(hrPrev) equals false, no operation is executed.) *)
	END_VAR

END_FUNCTION

// Functions/Basic Container Operations/F_VN_FillContainerExp/F_VN_FillContainerExp_TcVnRectangle_DINT

	{attribute 'TcIecLibraryType'}
	{attribute 'external_name' := 'F_VN_FillContainerExp_TcVnRectangle_DINT_GUID_17A9E6C5_773F_5847_5BFC_3012D0A2FCD6'}
	(* Partially fill the container with the specified value. Only possible for containers with basic elements. (expert function) *)
	FUNCTION F_VN_FillContainerExp_TcVnRectangle_DINT : HRESULT
	VAR_INPUT
		ipContainer	:	ITcVnContainer;	(* Container with basic elements *)
		stValue	:	REFERENCE TO TcVnRectangle_DINT;	(* Value to set the container elements *)
		nStartIdx	:	ULINT;	(* Start index *)
		nCount	:	ULINT;	(* Number of elements to set *)
		hrPrev	:	HRESULT;	(* HRESULT indicating the result of previous operations (If SUCCEEDED(hrPrev) equals false, no operation is executed.) *)
	END_VAR

END_FUNCTION

// Functions/Basic Container Operations/F_VN_FillContainerExp/F_VN_FillContainerExp_TcVnVector2_DINT

	{attribute 'TcIecLibraryType'}
	{attribute 'external_name' := 'F_VN_FillContainerExp_TcVnVector2_DINT_GUID_493BA62E_CDA0_5AF4_4E58_913A4C2EA5AF'}
	(* Partially fill the container with the specified value. Only possible for containers with basic elements. (expert function) *)
	FUNCTION F_VN_FillContainerExp_TcVnVector2_DINT : HRESULT
	VAR_INPUT
		ipContainer	:	ITcVnContainer;	(* Container with basic elements *)
		aValue	:	REFERENCE TO TcVnVector2_DINT;	(* Value to set the container elements *)
		nStartIdx	:	ULINT;	(* Start index *)
		nCount	:	ULINT;	(* Number of elements to set *)
		hrPrev	:	HRESULT;	(* HRESULT indicating the result of previous operations (If SUCCEEDED(hrPrev) equals false, no operation is executed.) *)
	END_VAR

END_FUNCTION

// Functions/Basic Container Operations/F_VN_FillContainerExp/F_VN_FillContainerExp_TcVnVector2_REAL

	{attribute 'TcIecLibraryType'}
	{attribute 'external_name' := 'F_VN_FillContainerExp_TcVnVector2_REAL_GUID_E5C621C9_CA59_5A04_79A7_BD2569534983'}
	(* Partially fill the container with the specified value. Only possible for containers with basic elements. (expert function) *)
	FUNCTION F_VN_FillContainerExp_TcVnVector2_REAL : HRESULT
	VAR_INPUT
		ipContainer	:	ITcVnContainer;	(* Container with basic elements *)
		aValue	:	REFERENCE TO TcVnVector2_REAL;	(* Value to set the container elements *)
		nStartIdx	:	ULINT;	(* Start index *)
		nCount	:	ULINT;	(* Number of elements to set *)
		hrPrev	:	HRESULT;	(* HRESULT indicating the result of previous operations (If SUCCEEDED(hrPrev) equals false, no operation is executed.) *)
	END_VAR

END_FUNCTION

// Functions/Basic Container Operations/F_VN_FillContainerExp/F_VN_FillContainerExp_TcVnVector3_REAL

	{attribute 'TcIecLibraryType'}
	{attribute 'external_name' := 'F_VN_FillContainerExp_TcVnVector3_REAL_GUID_6B0BC54E_4CCA_5442_7D50_D32DA2DA88D7'}
	(* Partially fill the container with the specified value. Only possible for containers with basic elements. (expert function) *)
	FUNCTION F_VN_FillContainerExp_TcVnVector3_REAL : HRESULT
	VAR_INPUT
		ipContainer	:	ITcVnContainer;	(* Container with basic elements *)
		aValue	:	REFERENCE TO TcVnVector3_REAL;	(* Value to set the container elements *)
		nStartIdx	:	ULINT;	(* Start index *)
		nCount	:	ULINT;	(* Number of elements to set *)
		hrPrev	:	HRESULT;	(* HRESULT indicating the result of previous operations (If SUCCEEDED(hrPrev) equals false, no operation is executed.) *)
	END_VAR

END_FUNCTION

// Functions/Basic Container Operations/F_VN_FillContainerExp/F_VN_FillContainerExp_TcVnVector4_DINT

	{attribute 'TcIecLibraryType'}
	{attribute 'external_name' := 'F_VN_FillContainerExp_TcVnVector4_DINT_GUID_4CA1BD05_C34B_5F32_702E_6C842E0E6CA6'}
	(* Partially fill the container with the specified value. Only possible for containers with basic elements. (expert function) *)
	FUNCTION F_VN_FillContainerExp_TcVnVector4_DINT : HRESULT
	VAR_INPUT
		ipContainer	:	ITcVnContainer;	(* Container with basic elements *)
		aValue	:	REFERENCE TO TcVnVector4_DINT;	(* Value to set the container elements *)
		nStartIdx	:	ULINT;	(* Start index *)
		nCount	:	ULINT;	(* Number of elements to set *)
		hrPrev	:	HRESULT;	(* HRESULT indicating the result of previous operations (If SUCCEEDED(hrPrev) equals false, no operation is executed.) *)
	END_VAR

END_FUNCTION

// Functions/Basic Container Operations/F_VN_FillContainerExp/F_VN_FillContainerExp_TcVnVector4_LREAL

	{attribute 'TcIecLibraryType'}
	{attribute 'external_name' := 'F_VN_FillContainerExp_TcVnVector4_LREAL_GUID_4284BC92_FBAD_57CE_60EF_853EAAAA5974'}
	(* Partially fill the container with the specified value. Only possible for containers with basic elements. (expert function) *)
	FUNCTION F_VN_FillContainerExp_TcVnVector4_LREAL : HRESULT
	VAR_INPUT
		ipContainer	:	ITcVnContainer;	(* Container with basic elements *)
		aValue	:	REFERENCE TO TcVnVector4_LREAL;	(* Value to set the container elements *)
		nStartIdx	:	ULINT;	(* Start index *)
		nCount	:	ULINT;	(* Number of elements to set *)
		hrPrev	:	HRESULT;	(* HRESULT indicating the result of previous operations (If SUCCEEDED(hrPrev) equals false, no operation is executed.) *)
	END_VAR

END_FUNCTION

// Functions/Basic Container Operations/F_VN_FillContainerExp/F_VN_FillContainerExp_UDINT

	{attribute 'TcIecLibraryType'}
	{attribute 'external_name' := 'F_VN_FillContainerExp_UDINT_GUID_5D9C5786_9DE6_5BEA_7A6B_236DD18DC857'}
	(* Partially fill the container with the specified value. Only possible for containers with basic elements. (expert function) *)
	FUNCTION F_VN_FillContainerExp_UDINT : HRESULT
	VAR_INPUT
		ipContainer	:	ITcVnContainer;	(* Container with basic elements *)
		nValue	:	UDINT;	(* Value to set the container elements *)
		nStartIdx	:	ULINT;	(* Start index *)
		nCount	:	ULINT;	(* Number of elements to set *)
		hrPrev	:	HRESULT;	(* HRESULT indicating the result of previous operations (If SUCCEEDED(hrPrev) equals false, no operation is executed.) *)
	END_VAR

END_FUNCTION

// Functions/Basic Container Operations/F_VN_FillContainerExp/F_VN_FillContainerExp_ULINT

	{attribute 'TcIecLibraryType'}
	{attribute 'external_name' := 'F_VN_FillContainerExp_ULINT_GUID_7D42DEA9_DDA6_5AB9_7BB0_6FD03818C6CD'}
	(* Partially fill the container with the specified value. Only possible for containers with basic elements. (expert function) *)
	FUNCTION F_VN_FillContainerExp_ULINT : HRESULT
	VAR_INPUT
		ipContainer	:	ITcVnContainer;	(* Container with basic elements *)
		nValue	:	ULINT;	(* Value to set the container elements *)
		nStartIdx	:	ULINT;	(* Start index *)
		nCount	:	ULINT;	(* Number of elements to set *)
		hrPrev	:	HRESULT;	(* HRESULT indicating the result of previous operations (If SUCCEEDED(hrPrev) equals false, no operation is executed.) *)
	END_VAR

END_FUNCTION

// Functions/Basic Container Operations/F_VN_GetAt/F_VN_GetAt_ITcVnContainer

	{attribute 'TcIecLibraryType'}
	{attribute 'external_name' := 'F_VN_GetAt_ITcVnContainer_GUID_984A7993_CFBC_58BA_60DF_8BED17F702F9'}
	(* Gets the ITcVnContainer element at the specified index of the source container. (Alternatively use interface method .GetAt.) *)
	FUNCTION F_VN_GetAt_ITcVnContainer : HRESULT
	VAR_INPUT
		ipSrcContainer	:	ITcVnContainer;	(* Container with ITcVnContainer elements *)
		ipDestContainer	:	REFERENCE TO ITcVnContainer;	(* Returns the container at the specified index *)
		nIndex	:	ULINT;	(* Index of the requested element *)
		hrPrev	:	HRESULT;	(* HRESULT indicating the result of previous operations (If SUCCEEDED(hrPrev) equals false, no operation is executed.) *)
	END_VAR

END_FUNCTION

// Functions/Basic Container Operations/F_VN_GetAt/F_VN_GetAt_DINT

	{attribute 'TcIecLibraryType'}
	{attribute 'external_name' := 'F_VN_GetAt_DINT_GUID_4FECF609_0716_5FAF_4BE4_AD8426C3C474'}
	(* Gets the DINT element at the specified index of the container. *)
	FUNCTION F_VN_GetAt_DINT : HRESULT
	VAR_INPUT
		ipContainer	:	ITcVnContainer;	(* Container with DINT elements *)
		nElement	:	REFERENCE TO DINT;	(* Returns the element at the specified index *)
		nIndex	:	ULINT;	(* Index of the requested element *)
		hrPrev	:	HRESULT;	(* HRESULT indicating the result of previous operations (If SUCCEEDED(hrPrev) equals false, no operation is executed.) *)
	END_VAR

END_FUNCTION

// Functions/Basic Container Operations/F_VN_GetAt/F_VN_GetAt_LREAL

	{attribute 'TcIecLibraryType'}
	{attribute 'external_name' := 'F_VN_GetAt_LREAL_GUID_4092A63B_BB5C_5AFB_5A6D_6BC903E97AD1'}
	(* Gets the LREAL element at the specified index of the container. *)
	FUNCTION F_VN_GetAt_LREAL : HRESULT
	VAR_INPUT
		ipContainer	:	ITcVnContainer;	(* Container with LREAL elements *)
		fElement	:	REFERENCE TO LREAL;	(* Returns the element at the specified index *)
		nIndex	:	ULINT;	(* Index of the requested element *)
		hrPrev	:	HRESULT;	(* HRESULT indicating the result of previous operations (If SUCCEEDED(hrPrev) equals false, no operation is executed.) *)
	END_VAR

END_FUNCTION

// Functions/Basic Container Operations/F_VN_GetAt/F_VN_GetAt_REAL

	{attribute 'TcIecLibraryType'}
	{attribute 'external_name' := 'F_VN_GetAt_REAL_GUID_82035886_E837_5FF4_4C2E_BA316678B433'}
	(* Gets the REAL element at the specified index of the container. *)
	FUNCTION F_VN_GetAt_REAL : HRESULT
	VAR_INPUT
		ipContainer	:	ITcVnContainer;	(* Container with REAL elements *)
		fElement	:	REFERENCE TO REAL;	(* Returns the element at the specified index *)
		nIndex	:	ULINT;	(* Index of the requested element *)
		hrPrev	:	HRESULT;	(* HRESULT indicating the result of previous operations (If SUCCEEDED(hrPrev) equals false, no operation is executed.) *)
	END_VAR

END_FUNCTION

// Functions/Basic Container Operations/F_VN_GetAt/F_VN_GetAt_SINT

	{attribute 'TcIecLibraryType'}
	{attribute 'external_name' := 'F_VN_GetAt_SINT_GUID_14038A4A_55C6_5C19_6B42_4B8543E667EB'}
	(* Gets the SINT element at the specified index of the container. *)
	FUNCTION F_VN_GetAt_SINT : HRESULT
	VAR_INPUT
		ipContainer	:	ITcVnContainer;	(* Container with SINT elements *)
		nElement	:	REFERENCE TO SINT;	(* Returns the element at the specified index *)
		nIndex	:	ULINT;	(* Index of the requested element *)
		hrPrev	:	HRESULT;	(* HRESULT indicating the result of previous operations (If SUCCEEDED(hrPrev) equals false, no operation is executed.) *)
	END_VAR

END_FUNCTION

// Functions/Basic Container Operations/F_VN_GetAt/F_VN_GetAt_TcVnDMatch

	{attribute 'TcIecLibraryType'}
	{attribute 'external_name' := 'F_VN_GetAt_TcVnDMatch_GUID_AE1225D9_2AD7_596B_4D8D_D472BF41DE94'}
	(* Gets the TcVnDMatch element at the specified index of the container. *)
	FUNCTION F_VN_GetAt_TcVnDMatch : HRESULT
	VAR_INPUT
		ipContainer	:	ITcVnContainer;	(* Container with TcVnDMatch elements *)
		stElement	:	REFERENCE TO TcVnDMatch;	(* Returns the element at the specified index *)
		nIndex	:	ULINT;	(* Index of the requested element *)
		hrPrev	:	HRESULT;	(* HRESULT indicating the result of previous operations (If SUCCEEDED(hrPrev) equals false, no operation is executed.) *)
	END_VAR

END_FUNCTION

// Functions/Basic Container Operations/F_VN_GetAt/F_VN_GetAt_TcVnKeyPoint

	{attribute 'TcIecLibraryType'}
	{attribute 'external_name' := 'F_VN_GetAt_TcVnKeyPoint_GUID_B110DEE4_56A9_5D79_51FD_7BF7E8D04135'}
	(* Gets the TcVnKeyPoint element at the specified index of the container. *)
	FUNCTION F_VN_GetAt_TcVnKeyPoint : HRESULT
	VAR_INPUT
		ipContainer	:	ITcVnContainer;	(* Container with TcVnKeyPoint elements *)
		stElement	:	REFERENCE TO TcVnKeyPoint;	(* Returns the element at the specified index *)
		nIndex	:	ULINT;	(* Index of the requested element *)
		hrPrev	:	HRESULT;	(* HRESULT indicating the result of previous operations (If SUCCEEDED(hrPrev) equals false, no operation is executed.) *)
	END_VAR

END_FUNCTION

// Functions/Basic Container Operations/F_VN_GetAt/F_VN_GetAt_TcVnPoint2_DINT

	{attribute 'TcIecLibraryType'}
	{attribute 'external_name' := 'F_VN_GetAt_TcVnPoint2_DINT_GUID_7F2BEC2B_1D00_5955_489F_24554E291091'}
	(* Gets the TcVnPoint2_DINT element at the specified index of the container. *)
	FUNCTION F_VN_GetAt_TcVnPoint2_DINT : HRESULT
	VAR_INPUT
		ipContainer	:	ITcVnContainer;	(* Container with TcVnPoint2_DINT elements *)
		aElement	:	REFERENCE TO TcVnPoint2_DINT;	(* Returns the element at the specified index *)
		nIndex	:	ULINT;	(* Index of the requested element *)
		hrPrev	:	HRESULT;	(* HRESULT indicating the result of previous operations (If SUCCEEDED(hrPrev) equals false, no operation is executed.) *)
	END_VAR

END_FUNCTION

// Functions/Basic Container Operations/F_VN_GetAt/F_VN_GetAt_TcVnPoint2_LREAL

	{attribute 'TcIecLibraryType'}
	{attribute 'external_name' := 'F_VN_GetAt_TcVnPoint2_LREAL_GUID_02FE9323_1EF4_5C4E_6AF2_7B38CA694696'}
	(* Gets the TcVnPoint2_LREAL element at the specified index of the container. *)
	FUNCTION F_VN_GetAt_TcVnPoint2_LREAL : HRESULT
	VAR_INPUT
		ipContainer	:	ITcVnContainer;	(* Container with TcVnPoint2_LREAL elements *)
		aElement	:	REFERENCE TO TcVnPoint2_LREAL;	(* Returns the element at the specified index *)
		nIndex	:	ULINT;	(* Index of the requested element *)
		hrPrev	:	HRESULT;	(* HRESULT indicating the result of previous operations (If SUCCEEDED(hrPrev) equals false, no operation is executed.) *)
	END_VAR

END_FUNCTION

// Functions/Basic Container Operations/F_VN_GetAt/F_VN_GetAt_TcVnPoint2_REAL

	{attribute 'TcIecLibraryType'}
	{attribute 'external_name' := 'F_VN_GetAt_TcVnPoint2_REAL_GUID_AB0B63A7_354D_56FF_7241_DEC5DBEA96F2'}
	(* Gets the TcVnPoint2_REAL element at the specified index of the container. *)
	FUNCTION F_VN_GetAt_TcVnPoint2_REAL : HRESULT
	VAR_INPUT
		ipContainer	:	ITcVnContainer;	(* Container with TcVnPoint2_REAL elements *)
		aElement	:	REFERENCE TO TcVnPoint2_REAL;	(* Returns the element at the specified index *)
		nIndex	:	ULINT;	(* Index of the requested element *)
		hrPrev	:	HRESULT;	(* HRESULT indicating the result of previous operations (If SUCCEEDED(hrPrev) equals false, no operation is executed.) *)
	END_VAR

END_FUNCTION

// Functions/Basic Container Operations/F_VN_GetAt/F_VN_GetAt_TcVnPoint3_LREAL

	{attribute 'TcIecLibraryType'}
	{attribute 'external_name' := 'F_VN_GetAt_TcVnPoint3_LREAL_GUID_0C2CC0BD_6743_5253_5C07_ED6782669908'}
	(* Gets the TcVnPoint3_LREAL element at the specified index of the container. *)
	FUNCTION F_VN_GetAt_TcVnPoint3_LREAL : HRESULT
	VAR_INPUT
		ipContainer	:	ITcVnContainer;	(* Container with TcVnPoint3_LREAL elements *)
		aElement	:	REFERENCE TO TcVnPoint3_LREAL;	(* Returns the element at the specified index *)
		nIndex	:	ULINT;	(* Index of the requested element *)
		hrPrev	:	HRESULT;	(* HRESULT indicating the result of previous operations (If SUCCEEDED(hrPrev) equals false, no operation is executed.) *)
	END_VAR

END_FUNCTION

// Functions/Basic Container Operations/F_VN_GetAt/F_VN_GetAt_TcVnPoint3_REAL

	{attribute 'TcIecLibraryType'}
	{attribute 'external_name' := 'F_VN_GetAt_TcVnPoint3_REAL_GUID_964802D3_245A_589B_4898_424205865D20'}
	(* Gets the TcVnPoint3_REAL element at the specified index of the container. *)
	FUNCTION F_VN_GetAt_TcVnPoint3_REAL : HRESULT
	VAR_INPUT
		ipContainer	:	ITcVnContainer;	(* Container with TcVnPoint3_REAL elements *)
		aElement	:	REFERENCE TO TcVnPoint3_REAL;	(* Returns the element at the specified index *)
		nIndex	:	ULINT;	(* Index of the requested element *)
		hrPrev	:	HRESULT;	(* HRESULT indicating the result of previous operations (If SUCCEEDED(hrPrev) equals false, no operation is executed.) *)
	END_VAR

END_FUNCTION

// Functions/Basic Container Operations/F_VN_GetAt/F_VN_GetAt_TcVnRectangle_DINT

	{attribute 'TcIecLibraryType'}
	{attribute 'external_name' := 'F_VN_GetAt_TcVnRectangle_DINT_GUID_E9A68DF9_B238_5F9D_4EC1_C0FC9E9B0531'}
	(* Gets the TcVnRectangle_DINT element at the specified index of the container. *)
	FUNCTION F_VN_GetAt_TcVnRectangle_DINT : HRESULT
	VAR_INPUT
		ipContainer	:	ITcVnContainer;	(* Container with TcVnRectangle_DINT elements *)
		stElement	:	REFERENCE TO TcVnRectangle_DINT;	(* Returns the element at the specified index *)
		nIndex	:	ULINT;	(* Index of the requested element *)
		hrPrev	:	HRESULT;	(* HRESULT indicating the result of previous operations (If SUCCEEDED(hrPrev) equals false, no operation is executed.) *)
	END_VAR

END_FUNCTION

// Functions/Basic Container Operations/F_VN_GetAt/F_VN_GetAt_TcVnVector2_DINT

	{attribute 'TcIecLibraryType'}
	{attribute 'external_name' := 'F_VN_GetAt_TcVnVector2_DINT_GUID_7BD77FC1_633C_54FA_66E9_F23B4C181C19'}
	(* Gets the TcVnVector2_DINT element at the specified index of the container. *)
	FUNCTION F_VN_GetAt_TcVnVector2_DINT : HRESULT
	VAR_INPUT
		ipContainer	:	ITcVnContainer;	(* Container with TcVnVector2_DINT elements *)
		aElement	:	REFERENCE TO TcVnVector2_DINT;	(* Returns the element at the specified index *)
		nIndex	:	ULINT;	(* Index of the requested element *)
		hrPrev	:	HRESULT;	(* HRESULT indicating the result of previous operations (If SUCCEEDED(hrPrev) equals false, no operation is executed.) *)
	END_VAR

END_FUNCTION

// Functions/Basic Container Operations/F_VN_GetAt/F_VN_GetAt_TcVnVector2_REAL

	{attribute 'TcIecLibraryType'}
	{attribute 'external_name' := 'F_VN_GetAt_TcVnVector2_REAL_GUID_0F5AC64C_EA53_5CBA_6EC0_871F55132C98'}
	(* Gets the TcVnVector2_REAL element at the specified index of the container. *)
	FUNCTION F_VN_GetAt_TcVnVector2_REAL : HRESULT
	VAR_INPUT
		ipContainer	:	ITcVnContainer;	(* Container with TcVnVector2_REAL elements *)
		aElement	:	REFERENCE TO TcVnVector2_REAL;	(* Returns the element at the specified index *)
		nIndex	:	ULINT;	(* Index of the requested element *)
		hrPrev	:	HRESULT;	(* HRESULT indicating the result of previous operations (If SUCCEEDED(hrPrev) equals false, no operation is executed.) *)
	END_VAR

END_FUNCTION

// Functions/Basic Container Operations/F_VN_GetAt/F_VN_GetAt_TcVnVector3_REAL

	{attribute 'TcIecLibraryType'}
	{attribute 'external_name' := 'F_VN_GetAt_TcVnVector3_REAL_GUID_734DF0C5_34D5_59F1_510F_A06D1060FC90'}
	(* Gets the TcVnVector3_REAL element at the specified index of the container. *)
	FUNCTION F_VN_GetAt_TcVnVector3_REAL : HRESULT
	VAR_INPUT
		ipContainer	:	ITcVnContainer;	(* Container with TcVnVector3_REAL elements *)
		aElement	:	REFERENCE TO TcVnVector3_REAL;	(* Returns the element at the specified index *)
		nIndex	:	ULINT;	(* Index of the requested element *)
		hrPrev	:	HRESULT;	(* HRESULT indicating the result of previous operations (If SUCCEEDED(hrPrev) equals false, no operation is executed.) *)
	END_VAR

END_FUNCTION

// Functions/Basic Container Operations/F_VN_GetAt/F_VN_GetAt_TcVnVector4_DINT

